LIN {X 0,Y 256.038,Z 225.896,A -85,B 0,C 180,E1 -18581.208,E2 -18581.208} C_VEL
LIN {X 0,Y 256.027,Z 225.882,A -85,B 0,C 180,E1 -18585.539,E2 -18585.539} C_VEL
LIN {X 0,Y 256.041,Z 225.899,A -85,B 0,C 180,E1 -18588.801,E2 -18588.801} C_VEL
LIN {X 0,Y 256.118,Z 225.896,A -85,B 0,C 180,E1 -18592.872,E2 -18592.872} C_VEL
LIN {X 0,Y 256.057,Z 225.889,A -85,B 0,C 180,E1 -18596.712,E2 -18596.712} C_VEL
LIN {X 0,Y 256.085,Z 225.887,A -85,B 0,C 180,E1 -18599.189,E2 -18599.189} C_VEL
LIN {X 0,Y 256.928,Z 228.457,A -85,B 0,C 180,E1 -18599.571,E2 -18599.571} C_VEL
LIN {X 0,Y 258.802,Z 230.64,A -85,B 0,C 180,E1 -18600.2,E2 -18600.2} C_VEL
LIN {X 0,Y 259.731,Z 231.462,A -85,B 0,C 180,E1 -18600.494,E2 -18600.494} C_VEL
LIN {X 0,Y 261.745,Z 234.708,A -85,B 0,C 180,E1 -18601.184,E2 -18601.184} C_VEL
LIN {X 0,Y 263.592,Z 236.729,A -85,B 0,C 180,E1 -18601.759,E2 -18601.759} C_VEL
LIN {X 0,Y 266.247,Z 240.339,A -85,B 0,C 180,E1 -18602.596,E2 -18602.596} C_VEL
LIN {X 0,Y 273.442,Z 250.412,A -85,B 0,C 180,E1 -18604.75,E2 -18604.75} C_VEL
LIN {X 0,Y 282.168,Z 263.234,A -85,B 0,C 180,E1 -18607.158,E2 -18607.158} C_VEL
LIN {X 0,Y 292.343,Z 279.507,A -85,B 0,C 180,E1 -18609.748,E2 -18609.748} C_VEL
LIN {X 0,Y 301.413,Z 295.689,A -85,B 0,C 180,E1 -18611.909,E2 -18611.909} C_VEL
LIN {X 0,Y 301.792,Z 296.477,A -85,B 0,C 180,E1 -18611.999,E2 -18611.999} C_VEL
LIN {X 0,Y 294.908,Z 420.321,A -85,B 0,C 180,E1 -18614.984,E2 -18614.984} C_VEL
LIN {X 0,Y 293.147,Z 437.641,A -85,B 0,C 180,E1 -18615.646,E2 -18615.646} C_VEL
LIN {X 0,Y 291.033,Z 452.968,A -85,B 0,C 180,E1 -18616.475,E2 -18616.475} C_VEL
LIN {X 0,Y 288.503,Z 467.873,A -85,B 0,C 180,E1 -18617.518,E2 -18617.518} C_VEL
LIN {X 0,Y 285.534,Z 482.731,A -85,B 0,C 180,E1 -18618.827,E2 -18618.827} C_VEL
LIN {X 0,Y 282.223,Z 496.554,A -85,B 0,C 180,E1 -18620.327,E2 -18620.327} C_VEL
LIN {X 0,Y 278.395,Z 510.812,A -85,B 0,C 180,E1 -18622.205,E2 -18622.205} C_VEL
LIN {X 0,Y 274.89,Z 522.936,A -85,B 0,C 180,E1 -18624.134,E2 -18624.134} C_VEL
LIN {X 0,Y 271.37,Z 534.312,A -85,B 0,C 180,E1 -18626.291,E2 -18626.291} C_VEL
LIN {X 0,Y 267.802,Z 545.342,A -85,B 0,C 180,E1 -18628.802,E2 -18628.802} C_VEL
LIN {X 0,Y 264.442,Z 555.354,A -85,B 0,C 180,E1 -18631.527,E2 -18631.527} C_VEL
LIN {X 0,Y 261.64,Z 563.721,A -85,B 0,C 180,E1 -18634.24,E2 -18634.24} C_VEL
LIN {X 0,Y 258.799,Z 572.627,A -85,B 0,C 180,E1 -18637.807,E2 -18637.807} C_VEL
LIN {X 0,Y 256.937,Z 579.031,A -85,B 0,C 180,E1 -18641.042,E2 -18641.042} C_VEL
LIN {X 0,Y 255.526,Z 584.251,A -85,B 0,C 180,E1 -18644.335,E2 -18644.335} C_VEL
LIN {X 0,Y 254.507,Z 588.356,A -85,B 0,C 180,E1 -18647.687,E2 -18647.687} C_VEL
LIN {X 0,Y 253.858,Z 591.244,A -85,B 0,C 180,E1 -18651.097,E2 -18651.097} C_VEL
LIN {X 0,Y 253.55,Z 593.058,A -85,B 0,C 180,E1 -18654.571,E2 -18654.571} C_VEL
LIN {X 0,Y 253.564,Z 593.757,A -85,B 0,C 180,E1 -18658.115,E2 -18658.115} C_VEL
LIN {X 0,Y 253.804,Z 593.171,A -85,B 0,C 180,E1 -18661.747,E2 -18661.747} C_VEL
LIN {X 0,Y 254.377,Z 591.318,A -85,B 0,C 180,E1 -18665.467,E2 -18665.467} C_VEL
LIN {X 0,Y 255.541,Z 588.082,A -85,B 0,C 180,E1 -18669.242,E2 -18669.242} C_VEL
LIN {X 0,Y 257.285,Z 583.305,A -85,B 0,C 180,E1 -18673.074,E2 -18673.074} C_VEL
LIN {X 0,Y 259.119,Z 578.582,A -85,B 0,C 180,E1 -18675.953,E2 -18675.953} C_VEL
LIN {X 0,Y 262.023,Z 571.463,A -85,B 0,C 180,E1 -18679.434,E2 -18679.434} C_VEL
LIN {X 0,Y 265.48,Z 563.42,A -85,B 0,C 180,E1 -18682.581,E2 -18682.581} C_VEL
LIN {X 0,Y 269.291,Z 554.393,A -85,B 0,C 180,E1 -18685.475,E2 -18685.475} C_VEL
LIN {X 0,Y 273.337,Z 544.565,A -85,B 0,C 180,E1 -18688.051,E2 -18688.051} C_VEL
LIN {X 0,Y 277.708,Z 533.552,A -85,B 0,C 180,E1 -18690.454,E2 -18690.454} C_VEL
LIN {X 0,Y 282.075,Z 521.913,A -85,B 0,C 180,E1 -18692.578,E2 -18692.578} C_VEL
LIN {X 0,Y 286.394,Z 509.229,A -85,B 0,C 180,E1 -18694.499,E2 -18694.499} C_VEL
LIN {X 0,Y 290.638,Z 495.548,A -85,B 0,C 180,E1 -18696.193,E2 -18696.193} C_VEL
LIN {X 0,Y 294.579,Z 480.888,A -85,B 0,C 180,E1 -18697.688,E2 -18697.688} C_VEL
LIN {X 0,Y 298.07,Z 466.156,A -85,B 0,C 180,E1 -18698.882,E2 -18698.882} C_VEL
LIN {X 0,Y 301.12,Z 449.617,A -85,B 0,C 180,E1 -18699.957,E2 -18699.957} C_VEL
LIN {X 0,Y 303.68,Z 432.171,A -85,B 0,C 180,E1 -18700.764,E2 -18700.764} C_VEL
LIN {X 0,Y 305.378,Z 415.089,A -85,B 0,C 180,E1 -18701.291,E2 -18701.291} C_VEL
LIN {X 0,Y 306.012,Z 404.805,A -85,B 0,C 180,E1 -18701.555,E2 -18701.555} C_VEL
LIN {X 0,Y 305.769,Z 400.957,A -85,B 0,C 180,E1 -18701.757,E2 -18701.757} C_VEL
LIN {X 0,Y 302.881,Z 389.177,A -85,B 0,C 180,E1 -18702.878,E2 -18702.878} C_VEL
LIN {X 0,Y 302.776,Z 385.325,A -85,B 0,C 180,E1 -18703.057,E2 -18703.057} C_VEL
LIN {X 0,Y 308.251,Z 305.412,A -85,B 0,C 180,E1 -18704.992,E2 -18704.992} C_VEL
LIN {X 0,Y 302.68,Z 295.118,A -85,B 0,C 180,E1 -18706.932,E2 -18706.932} C_VEL
LIN {X 0,Y 297.182,Z 285.913,A -85,B 0,C 180,E1 -18709.029,E2 -18709.029} C_VEL
LIN {X 0,Y 292.134,Z 278.185,A -85,B 0,C 180,E1 -18711.157,E2 -18711.157} C_VEL
LIN {X 0,Y 288.761,Z 273.365,A -85,B 0,C 180,E1 -18712.725,E2 -18712.725} C_VEL
LIN {X 0,Y 286.101,Z 269.539,A -85,B 0,C 180,E1 -18714.079,E2 -18714.079} C_VEL
LIN {X 0,Y 283.274,Z 265.593,A -85,B 0,C 180,E1 -18715.636,E2 -18715.636} C_VEL
LIN {X 0,Y 280.468,Z 261.788,A -85,B 0,C 180,E1 -18717.378,E2 -18717.378} C_VEL
LIN {X 0,Y 277.317,Z 257.984,A -85,B 0,C 180,E1 -18719.571,E2 -18719.571} C_VEL
LIN {X 0,Y 276.388,Z 256.203,A -85,B 0,C 180,E1 -18720.363,E2 -18720.363} C_VEL
LIN {X 0,Y 273.687,Z 253.629,A -85,B 0,C 180,E1 -18722.755,E2 -18722.755} C_VEL
LIN {X 0,Y 272.252,Z 251.029,A -85,B 0,C 180,E1 -18724.441,E2 -18724.441} C_VEL
LIN {X 0,Y 268.845,Z 248.558,A -85,B 0,C 180,E1 -18730.543,E2 -18730.543} C_VEL
LIN {X 0,Y 268.488,Z 248.039,A -85,B 0,C 180,E1 -18733.625,E2 -18733.625} C_VEL
LIN {X 0,Y 269.382,Z 249.399,A -85,B 0,C 180,E1 -18737.862,E2 -18737.862} C_VEL
LIN {X 0,Y 272.037,Z 251.261,A -85,B 0,C 180,E1 -18741.994,E2 -18741.994} C_VEL
LIN {X 0,Y 273.82,Z 254.481,A -85,B 0,C 180,E1 -18744.088,E2 -18744.088} C_VEL
LIN {X 0,Y 276.278,Z 256.688,A -85,B 0,C 180,E1 -18746.239,E2 -18746.239} C_VEL
LIN {X 0,Y 278.589,Z 260.18,A -85,B 0,C 180,E1 -18748.044,E2 -18748.044} C_VEL
LIN {X 0,Y 280.384,Z 262.136,A -85,B 0,C 180,E1 -18749.233,E2 -18749.233} C_VEL
LIN {X 0,Y 285.039,Z 268.873,A -85,B 0,C 180,E1 -18752.04,E2 -18752.04} C_VEL
LIN {X 0,Y 289.206,Z 275.406,A -85,B 0,C 180,E1 -18754.208,E2 -18754.208} C_VEL
LIN {X 0,Y 293.992,Z 283.483,A -85,B 0,C 180,E1 -18756.42,E2 -18756.42} C_VEL
LIN {X 0,Y 299.014,Z 292.67,A -85,B 0,C 180,E1 -18758.503,E2 -18758.503} C_VEL
LIN {X 0,Y 304.296,Z 303.274,A -85,B 0,C 180,E1 -18760.508,E2 -18760.508} C_VEL
LIN {X 0,Y 308.003,Z 311.578,A -85,B 0,C 180,E1 -18761.836,E2 -18761.836} C_VEL
LIN {X 0,Y 299.594,Z 433.298,A -85,B 0,C 180,E1 -18764.803,E2 -18764.803} C_VEL
LIN {X 0,Y 297.272,Z 451.036,A -85,B 0,C 180,E1 -18765.45,E2 -18765.45} C_VEL
LIN {X 0,Y 294.278,Z 467.286,A -85,B 0,C 180,E1 -18766.281,E2 -18766.281} C_VEL
LIN {X 0,Y 290.622,Z 483.374,A -85,B 0,C 180,E1 -18767.379,E2 -18767.379} C_VEL
LIN {X 0,Y 286.484,Z 498.911,A -85,B 0,C 180,E1 -18768.751,E2 -18768.751} C_VEL
LIN {X 0,Y 282.022,Z 513.293,A -85,B 0,C 180,E1 -18770.312,E2 -18770.312} C_VEL
LIN {X 0,Y 277.311,Z 527.146,A -85,B 0,C 180,E1 -18772.179,E2 -18772.179} C_VEL
LIN {X 0,Y 272.824,Z 538.984,A -85,B 0,C 180,E1 -18774.12,E2 -18774.12} C_VEL
LIN {X 0,Y 267.857,Z 551.328,A -85,B 0,C 180,E1 -18776.562,E2 -18776.562} C_VEL
LIN {X 0,Y 263.501,Z 561.999,A -85,B 0,C 180,E1 -18779.137,E2 -18779.137} C_VEL
LIN {X 0,Y 259.085,Z 572.215,A -85,B 0,C 180,E1 -18782.097,E2 -18782.097} C_VEL
LIN {X 0,Y 254.995,Z 581.851,A -85,B 0,C 180,E1 -18785.577,E2 -18785.577} C_VEL
LIN {X 0,Y 251.539,Z 590.511,A -85,B 0,C 180,E1 -18789.555,E2 -18789.555} C_VEL
LIN {X 0,Y 249.159,Z 597.289,A -85,B 0,C 180,E1 -18793.613,E2 -18793.613} C_VEL
LIN {X 0,Y 247.861,Z 601.425,A -85,B 0,C 180,E1 -18796.886,E2 -18796.886} C_VEL
LIN {X 0,Y 247.112,Z 604.608,A -85,B 0,C 180,E1 -18800.171,E2 -18800.171} C_VEL
LIN {X 0,Y 246.859,Z 606.706,A -85,B 0,C 180,E1 -18803.457,E2 -18803.457} C_VEL
LIN {X 0,Y 246.839,Z 607.901,A -85,B 0,C 180,E1 -18806.732,E2 -18806.732} C_VEL
LIN {X 0,Y 246.982,Z 608.041,A -85,B 0,C 180,E1 -18809.996,E2 -18809.996} C_VEL
LIN {X 0,Y 246.867,Z 607.256,A -85,B 0,C 180,E1 -18813.26,E2 -18813.26} C_VEL
LIN {X 0,Y 246.908,Z 606.416,A -85,B 0,C 180,E1 -18814.977,E2 -18814.977} C_VEL
LIN {X 0,Y 246.951,Z 604.091,A -85,B 0,C 180,E1 -18818.176,E2 -18818.176} C_VEL
LIN {X 0,Y 247.356,Z 600.725,A -85,B 0,C 180,E1 -18821.467,E2 -18821.467} C_VEL
LIN {X 0,Y 248.35,Z 596.177,A -85,B 0,C 180,E1 -18824.751,E2 -18824.751} C_VEL
LIN {X 0,Y 249.763,Z 590.504,A -85,B 0,C 180,E1 -18828.026,E2 -18828.026} C_VEL
LIN {X 0,Y 251.845,Z 583.51,A -85,B 0,C 180,E1 -18831.266,E2 -18831.266} C_VEL
LIN {X 0,Y 254.487,Z 575.039,A -85,B 0,C 180,E1 -18834.467,E2 -18834.467} C_VEL
LIN {X 0,Y 257.909,Z 564.935,A -85,B 0,C 180,E1 -18837.592,E2 -18837.592} C_VEL
LIN {X 0,Y 261.447,Z 554.509,A -85,B 0,C 180,E1 -18840.261,E2 -18840.261} C_VEL
LIN {X 0,Y 264.867,Z 544.091,A -85,B 0,C 180,E1 -18842.495,E2 -18842.495} C_VEL
LIN {X 0,Y 268.706,Z 531.999,A -85,B 0,C 180,E1 -18844.666,E2 -18844.666} C_VEL
LIN {X 0,Y 272.764,Z 518.677,A -85,B 0,C 180,E1 -18846.641,E2 -18846.641} C_VEL
LIN {X 0,Y 276.338,Z 505.257,A -85,B 0,C 180,E1 -18848.304,E2 -18848.304} C_VEL
LIN {X 0,Y 280.028,Z 490.239,A -85,B 0,C 180,E1 -18849.784,E2 -18849.784} C_VEL
LIN {X 0,Y 283.164,Z 474.912,A -85,B 0,C 180,E1 -18851.002,E2 -18851.002} C_VEL
LIN {X 0,Y 285.87,Z 458.777,A -85,B 0,C 180,E1 -18851.996,E2 -18851.996} C_VEL
LIN {X 0,Y 288.082,Z 442.453,A -85,B 0,C 180,E1 -18852.721,E2 -18852.721} C_VEL
LIN {X 0,Y 289.436,Z 426.385,A -85,B 0,C 180,E1 -18853.222,E2 -18853.222} C_VEL
LIN {X 0,Y 296.146,Z 306.323,A -85,B 0,C 180,E1 -18856.146,E2 -18856.146} C_VEL
LIN {X 0,Y 288.318,Z 289.97,A -85,B 0,C 180,E1 -18858.143,E2 -18858.143} C_VEL
LIN {X 0,Y 280.841,Z 275.817,A -85,B 0,C 180,E1 -18860.152,E2 -18860.152} C_VEL
LIN {X 0,Y 272.784,Z 261.806,A -85,B 0,C 180,E1 -18862.449,E2 -18862.449} C_VEL
LIN {X 0,Y 263.31,Z 246.71,A -85,B 0,C 180,E1 -18865.389,E2 -18865.389} C_VEL
LIN {X 0,Y 259.388,Z 241.321,A -85,B 0,C 180,E1 -18866.667,E2 -18866.667} C_VEL
LIN {X 0,Y 256.72,Z 237.707,A -85,B 0,C 180,E1 -18867.574,E2 -18867.574} C_VEL
LIN {X 0,Y 253.409,Z 233.62,A -85,B 0,C 180,E1 -18868.726,E2 -18868.726} C_VEL
LIN {X 0,Y 252.392,Z 231.94,A -85,B 0,C 180,E1 -18869.11,E2 -18869.11} C_VEL
LIN {X 0,Y 250.174,Z 229.865,A -85,B 0,C 180,E1 -18869.889,E2 -18869.889} C_VEL
LIN {X 0,Y 249.156,Z 227.398,A -85,B 0,C 180,E1 -18870.335,E2 -18870.335} C_VEL
LIN {X 0,Y 249.056,Z 226.774,A -85,B 0,C 180,E1 -18870.427,E2 -18870.427} C_VEL
LIN {X 0,Y 249.129,Z 226.741,A -85,B 0,C 180,E1 -18874.967,E2 -18874.967} C_VEL
LIN {X 0,Y 249.109,Z 226.742,A -85,B 0,C 180,E1 -18878.577,E2 -18878.577} C_VEL
LIN {X 0,Y 249.217,Z 226.755,A -85,B 0,C 180,E1 -18883.621,E2 -18883.621} C_VEL
LIN {X 0,Y 249.226,Z 226.706,A -85,B 0,C 180,E1 -18888.616,E2 -18888.616} C_VEL
LIN {X 0,Y 249.453,Z 226.725,A -85,B 0,C 180,E1 -18891.903,E2 -18891.903} C_VEL
LIN {X 0,Y 249.406,Z 226.675,A -85,B 0,C 180,E1 -18896.77,E2 -18896.77} C_VEL
LIN {X 0,Y 249.701,Z 226.689,A -85,B 0,C 180,E1 -18900.001,E2 -18900.001} C_VEL
LIN {X 0,Y 249.406,Z 226.706,A -85,B 0,C 180,E1 -18903.232,E2 -18903.232} C_VEL
LIN {X 0,Y 249.411,Z 226.715,A -85,B 0,C 180,E1 -18906.78,E2 -18906.78} C_VEL
LIN {X 0,Y 249.318,Z 226.724,A -85,B 0,C 180,E1 -18909.738,E2 -18909.738} C_VEL
LIN {X 0,Y 249.176,Z 226.755,A -85,B 0,C 180,E1 -18914.706,E2 -18914.706} C_VEL
LIN {X 0,Y 249.115,Z 226.735,A -85,B 0,C 180,E1 -18918.08,E2 -18918.08} C_VEL
LIN {X 0,Y 249.065,Z 226.767,A -85,B 0,C 180,E1 -18921.521,E2 -18921.521} C_VEL
LIN {X 0,Y 249.109,Z 226.736,A -85,B 0,C 180,E1 -18925.485,E2 -18925.485} C_VEL
LIN {X 0,Y 249.063,Z 226.773,A -85,B 0,C 180,E1 -18928.997,E2 -18928.997} C_VEL
LIN {X 0,Y 249.011,Z 226.751,A -85,B 0,C 180,E1 -18932.43,E2 -18932.43} C_VEL
LIN {X 0,Y 249.029,Z 226.778,A -85,B 0,C 180,E1 -18936.347,E2 -18936.347} C_VEL
LIN {X 0,Y 248.976,Z 226.764,A -85,B 0,C 180,E1 -18940.485,E2 -18940.485} C_VEL
LIN {X 0,Y 248.986,Z 226.782,A -85,B 0,C 180,E1 -18942.795,E2 -18942.795} C_VEL
LIN {X 0,Y 248.996,Z 226.78,A -85,B 0,C 180,E1 -18947.366,E2 -18947.366} C_VEL
LIN {X 0,Y 249.032,Z 226.769,A -85,B 0,C 180,E1 -18952.205,E2 -18952.205} C_VEL
LIN {X 0,Y 249.031,Z 226.763,A -85,B 0,C 180,E1 -18956.618,E2 -18956.618} C_VEL
LIN {X 0,Y 249.009,Z 226.772,A -85,B 0,C 180,E1 -18957.093,E2 -18957.093} C_VEL
LIN {X 0,Y 249.907,Z 229.476,A -85,B 0,C 180,E1 -18957.532,E2 -18957.532} C_VEL
LIN {X 0,Y 251.995,Z 231.702,A -85,B 0,C 180,E1 -18958.28,E2 -18958.28} C_VEL
LIN {X 0,Y 252.914,Z 232.566,A -85,B 0,C 180,E1 -18958.598,E2 -18958.598} C_VEL
LIN {X 0,Y 254.905,Z 235.733,A -85,B 0,C 180,E1 -18959.339,E2 -18959.339} C_VEL
LIN {X 0,Y 256.628,Z 237.548,A -85,B 0,C 180,E1 -18959.919,E2 -18959.919} C_VEL
LIN {X 0,Y 259.169,Z 241.121,A -85,B 0,C 180,E1 -18960.789,E2 -18960.789} C_VEL
LIN {X 0,Y 260.595,Z 242.915,A -85,B 0,C 180,E1 -18961.253,E2 -18961.253} C_VEL
LIN {X 0,Y 267.808,Z 252.881,A -85,B 0,C 180,E1 -18963.525,E2 -18963.525} C_VEL
LIN {X 0,Y 277.279,Z 266.774,A -85,B 0,C 180,E1 -18966.261,E2 -18966.261} C_VEL
LIN {X 0,Y 287.941,Z 283.964,A -85,B 0,C 180,E1 -18969.081,E2 -18969.081} C_VEL
LIN {X 0,Y 296.28,Z 298.863,A -85,B 0,C 180,E1 -18971.129,E2 -18971.129} C_VEL
LIN {X 0,Y 289.398,Z 420.084,A -85,B 0,C 180,E1 -18974.104,E2 -18974.104} C_VEL
LIN {X 0,Y 287.7,Z 436.638,A -85,B 0,C 180,E1 -18974.734,E2 -18974.734} C_VEL
LIN {X 0,Y 285.512,Z 452.308,A -85,B 0,C 180,E1 -18975.572,E2 -18975.572} C_VEL
LIN {X 0,Y 282.695,Z 468.412,A -85,B 0,C 180,E1 -18976.709,E2 -18976.709} C_VEL
LIN {X 0,Y 279.498,Z 483.759,A -85,B 0,C 180,E1 -18978.093,E2 -18978.093} C_VEL
LIN {X 0,Y 276.228,Z 496.992,A -85,B 0,C 180,E1 -18979.56,E2 -18979.56} C_VEL
LIN {X 0,Y 272.277,Z 511.211,A -85,B 0,C 180,E1 -18981.469,E2 -18981.469} C_VEL
LIN {X 0,Y 268.088,Z 524.98,A -85,B 0,C 180,E1 -18983.734,E2 -18983.734} C_VEL
LIN {X 0,Y 264.114,Z 537.241,A -85,B 0,C 180,E1 -18986.189,E2 -18986.189} C_VEL
LIN {X 0,Y 260.375,Z 548.339,A -85,B 0,C 180,E1 -18988.873,E2 -18988.873} C_VEL
LIN {X 0,Y 256.717,Z 558.837,A -85,B 0,C 180,E1 -18991.965,E2 -18991.965} C_VEL
LIN {X 0,Y 253.366,Z 568.512,A -85,B 0,C 180,E1 -18995.495,E2 -18995.495} C_VEL
LIN {X 0,Y 250.967,Z 575.869,A -85,B 0,C 180,E1 -18998.864,E2 -18998.864} C_VEL
LIN {X 0,Y 249.226,Z 581.744,A -85,B 0,C 180,E1 -19002.213,E2 -19002.213} C_VEL
LIN {X 0,Y 248.035,Z 586.383,A -85,B 0,C 180,E1 -19005.55,E2 -19005.55} C_VEL
LIN {X 0,Y 247.278,Z 589.203,A -85,B 0,C 180,E1 -19008.222,E2 -19008.222} C_VEL
LIN {X 0,Y 246.668,Z 591.951,A -85,B 0,C 180,E1 -19011.743,E2 -19011.743} C_VEL
LIN {X 0,Y 246.429,Z 593.489,A -85,B 0,C 180,E1 -19015.331,E2 -19015.331} C_VEL
LIN {X 0,Y 246.496,Z 593.914,A -85,B 0,C 180,E1 -19018.996,E2 -19018.996} C_VEL
LIN {X 0,Y 246.813,Z 593.149,A -85,B 0,C 180,E1 -19022.757,E2 -19022.757} C_VEL
LIN {X 0,Y 247.57,Z 591.009,A -85,B 0,C 180,E1 -19026.598,E2 -19026.598} C_VEL
LIN {X 0,Y 248.959,Z 587.441,A -85,B 0,C 180,E1 -19030.49,E2 -19030.49} C_VEL
LIN {X 0,Y 250.174,Z 584.29,A -85,B 0,C 180,E1 -19033.078,E2 -19033.078} C_VEL
LIN {X 0,Y 252.3,Z 579.106,A -85,B 0,C 180,E1 -19036.41,E2 -19036.41} C_VEL
LIN {X 0,Y 255.24,Z 572.41,A -85,B 0,C 180,E1 -19039.829,E2 -19039.829} C_VEL
LIN {X 0,Y 258.535,Z 565.201,A -85,B 0,C 180,E1 -19042.801,E2 -19042.801} C_VEL
LIN {X 0,Y 262.429,Z 556.354,A -85,B 0,C 180,E1 -19045.778,E2 -19045.778} C_VEL
LIN {X 0,Y 266.526,Z 547.015,A -85,B 0,C 180,E1 -19048.381,E2 -19048.381} C_VEL
LIN {X 0,Y 270.957,Z 536.584,A -85,B 0,C 180,E1 -19050.81,E2 -19050.81} C_VEL
LIN {X 0,Y 275.696,Z 524.377,A -85,B 0,C 180,E1 -19053.156,E2 -19053.156} C_VEL
LIN {X 0,Y 280.55,Z 511.023,A -85,B 0,C 180,E1 -19055.246,E2 -19055.246} C_VEL
LIN {X 0,Y 284.791,Z 498.12,A -85,B 0,C 180,E1 -19056.909,E2 -19056.909} C_VEL
LIN {X 0,Y 288.97,Z 483.644,A -85,B 0,C 180,E1 -19058.454,E2 -19058.454} C_VEL
LIN {X 0,Y 292.841,Z 468.101,A -85,B 0,C 180,E1 -19059.769,E2 -19059.769} C_VEL
LIN {X 0,Y 295.961,Z 452.361,A -85,B 0,C 180,E1 -19060.821,E2 -19060.821} C_VEL
LIN {X 0,Y 298.537,Z 435.936,A -85,B 0,C 180,E1 -19061.641,E2 -19061.641} C_VEL
LIN {X 0,Y 300.516,Z 418.44,A -85,B 0,C 180,E1 -19062.234,E2 -19062.234} C_VEL
LIN {X 0,Y 302.776,Z 385.325,A -85,B 0,C 180,E1 -19063.057,E2 -19063.057} C_VEL
LIN {X 0,Y 302.834,Z 379.541,A -85,B 0,C 180,E1 -19063.278,E2 -19063.278} C_VEL
LIN {X 0,Y 301.699,Z 370.313,A -85,B 0,C 180,E1 -19063.936,E2 -19063.936} C_VEL
LIN {X 0,Y 300.552,Z 361.092,A -85,B 0,C 180,E1 -19064.612,E2 -19064.612} C_VEL
LIN {X 0,Y 300.563,Z 355.31,A -85,B 0,C 180,E1 -19064.855,E2 -19064.855} C_VEL
LIN {X 0,Y 303.884,Z 308.521,A -85,B 0,C 180,E1 -19066.007,E2 -19066.007} C_VEL
LIN {X 0,Y 298.074,Z 297.794,A -85,B 0,C 180,E1 -19068.171,E2 -19068.171} C_VEL
LIN {X 0,Y 293.131,Z 289.563,A -85,B 0,C 180,E1 -19070.187,E2 -19070.187} C_VEL
LIN {X 0,Y 289.122,Z 283.386,A -85,B 0,C 180,E1 -19071.983,E2 -19071.983} C_VEL
LIN {X 0,Y 284.509,Z 276.454,A -85,B 0,C 180,E1 -19074.329,E2 -19074.329} C_VEL
LIN {X 0,Y 281.361,Z 272.03,A -85,B 0,C 180,E1 -19076.125,E2 -19076.125} C_VEL
LIN {X 0,Y 278.07,Z 267.628,A -85,B 0,C 180,E1 -19078.261,E2 -19078.261} C_VEL
LIN {X 0,Y 275.471,Z 264.089,A -85,B 0,C 180,E1 -19080.228,E2 -19080.228} C_VEL
LIN {X 0,Y 274.706,Z 262.786,A -85,B 0,C 180,E1 -19080.915,E2 -19080.915} C_VEL
LIN {X 0,Y 272.3,Z 260.326,A -85,B 0,C 180,E1 -19083.154,E2 -19083.154} C_VEL
LIN {X 0,Y 271.101,Z 258.011,A -85,B 0,C 180,E1 -19084.646,E2 -19084.646} C_VEL
LIN {X 0,Y 267.875,Z 255.592,A -85,B 0,C 180,E1 -19090.582,E2 -19090.582} C_VEL
LIN {X 0,Y 267.54,Z 255.058,A -85,B 0,C 180,E1 -19093.675,E2 -19093.675} C_VEL
LIN {X 0,Y 269.01,Z 256.997,A -85,B 0,C 180,E1 -19099.06,E2 -19099.06} C_VEL
LIN {X 0,Y 270.831,Z 258.241,A -85,B 0,C 180,E1 -19101.721,E2 -19101.721} C_VEL
LIN {X 0,Y 272.644,Z 261.462,A -85,B 0,C 180,E1 -19103.918,E2 -19103.918} C_VEL
LIN {X 0,Y 274.806,Z 263.495,A -85,B 0,C 180,E1 -19105.865,E2 -19105.865} C_VEL
LIN {X 0,Y 277.37,Z 267.233,A -85,B 0,C 180,E1 -19107.919,E2 -19107.919} C_VEL
LIN {X 0,Y 278.726,Z 268.794,A -85,B 0,C 180,E1 -19108.842,E2 -19108.842} C_VEL
LIN {X 0,Y 283.026,Z 275.276,A -85,B 0,C 180,E1 -19111.553,E2 -19111.553} C_VEL
LIN {X 0,Y 287.145,Z 281.958,A -85,B 0,C 180,E1 -19113.772,E2 -19113.772} C_VEL
LIN {X 0,Y 291.968,Z 290.428,A -85,B 0,C 180,E1 -19116.085,E2 -19116.085} C_VEL
LIN {X 0,Y 297.475,Z 300.983,A -85,B 0,C 180,E1 -19118.432,E2 -19118.432} C_VEL
LIN {X 0,Y 302.651,Z 312.143,A -85,B 0,C 180,E1 -19120.45,E2 -19120.45} C_VEL
LIN {X 0,Y 303.684,Z 314.617,A -85,B 0,C 180,E1 -19120.838,E2 -19120.838} C_VEL
LIN {X 0,Y 295.081,Z 433.216,A -85,B 0,C 180,E1 -19123.744,E2 -19123.744} C_VEL
LIN {X 0,Y 292.778,Z 450.274,A -85,B 0,C 180,E1 -19124.364,E2 -19124.364} C_VEL
LIN {X 0,Y 289.776,Z 466.339,A -85,B 0,C 180,E1 -19125.179,E2 -19125.179} C_VEL
LIN {X 0,Y 285.978,Z 482.599,A -85,B 0,C 180,E1 -19126.274,E2 -19126.274} C_VEL
LIN {X 0,Y 282.19,Z 496.689,A -85,B 0,C 180,E1 -19127.5,E2 -19127.5} C_VEL
LIN {X 0,Y 277.537,Z 511.374,A -85,B 0,C 180,E1 -19129.061,E2 -19129.061} C_VEL
LIN {X 0,Y 272.87,Z 524.548,A -85,B 0,C 180,E1 -19130.81,E2 -19130.81} C_VEL
LIN {X 0,Y 267.863,Z 537.438,A -85,B 0,C 180,E1 -19132.879,E2 -19132.879} C_VEL
LIN {X 0,Y 263.374,Z 548.377,A -85,B 0,C 180,E1 -19134.987,E2 -19134.987} C_VEL
LIN {X 0,Y 258.621,Z 559.277,A -85,B 0,C 180,E1 -19137.535,E2 -19137.535} C_VEL
LIN {X 0,Y 254.368,Z 568.668,A -85,B 0,C 180,E1 -19140.174,E2 -19140.174} C_VEL
LIN {X 0,Y 250.23,Z 577.854,A -85,B 0,C 180,E1 -19143.293,E2 -19143.293} C_VEL
LIN {X 0,Y 246.892,Z 585.568,A -85,B 0,C 180,E1 -19146.511,E2 -19146.511} C_VEL
LIN {X 0,Y 244.201,Z 591.949,A -85,B 0,C 180,E1 -19149.793,E2 -19149.793} C_VEL
LIN {X 0,Y 242.221,Z 597.355,A -85,B 0,C 180,E1 -19153.231,E2 -19153.231} C_VEL
LIN {X 0,Y 240.88,Z 601.326,A -85,B 0,C 180,E1 -19156.498,E2 -19156.498} C_VEL
LIN {X 0,Y 240.049,Z 604.468,A -85,B 0,C 180,E1 -19159.879,E2 -19159.879} C_VEL
LIN {X 0,Y 239.77,Z 606.548,A -85,B 0,C 180,E1 -19163.263,E2 -19163.263} C_VEL
LIN {X 0,Y 239.744,Z 607.704,A -85,B 0,C 180,E1 -19166.635,E2 -19166.635} C_VEL
LIN {X 0,Y 239.912,Z 607.825,A -85,B 0,C 180,E1 -19169.996,E2 -19169.996} C_VEL
LIN {X 0,Y 239.773,Z 606.999,A -85,B 0,C 180,E1 -19173.357,E2 -19173.357} C_VEL
LIN {X 0,Y 239.817,Z 606.2,A -85,B 0,C 180,E1 -19175.04,E2 -19175.04} C_VEL
LIN {X 0,Y 239.869,Z 603.79,A -85,B 0,C 180,E1 -19178.42,E2 -19178.42} C_VEL
LIN {X 0,Y 240.328,Z 600.398,A -85,B 0,C 180,E1 -19181.808,E2 -19181.808} C_VEL
LIN {X 0,Y 241.667,Z 594.763,A -85,B 0,C 180,E1 -19185.876,E2 -19185.876} C_VEL
LIN {X 0,Y 243.368,Z 588.425,A -85,B 0,C 180,E1 -19189.391,E2 -19189.391} C_VEL
LIN {X 0,Y 245.761,Z 581.043,A -85,B 0,C 180,E1 -19192.704,E2 -19192.704} C_VEL
LIN {X 0,Y 248.755,Z 572.18,A -85,B 0,C 180,E1 -19195.966,E2 -19195.966} C_VEL
LIN {X 0,Y 252.554,Z 561.576,A -85,B 0,C 180,E1 -19199.137,E2 -19199.137} C_VEL
LIN {X 0,Y 256.203,Z 550.95,A -85,B 0,C 180,E1 -19201.749,E2 -19201.749} C_VEL
LIN {X 0,Y 260.116,Z 539.507,A -85,B 0,C 180,E1 -19204.094,E2 -19204.094} C_VEL
LIN {X 0,Y 264.255,Z 526.727,A -85,B 0,C 180,E1 -19206.275,E2 -19206.275} C_VEL
LIN {X 0,Y 268.286,Z 513.067,A -85,B 0,C 180,E1 -19208.199,E2 -19208.199} C_VEL
LIN {X 0,Y 272.426,Z 497.808,A -85,B 0,C 180,E1 -19209.914,E2 -19209.914} C_VEL
LIN {X 0,Y 275.764,Z 483.143,A -85,B 0,C 180,E1 -19211.25,E2 -19211.25} C_VEL
LIN {X 0,Y 278.855,Z 467.321,A -85,B 0,C 180,E1 -19212.384,E2 -19212.384} C_VEL
LIN {X 0,Y 281.427,Z 451.327,A -85,B 0,C 180,E1 -19213.244,E2 -19213.244} C_VEL
LIN {X 0,Y 283.433,Z 434.03,A -85,B 0,C 180,E1 -19213.902,E2 -19213.902} C_VEL
LIN {X 0,Y 290.792,Z 308.784,A -85,B 0,C 180,E1 -19217.015,E2 -19217.015} C_VEL
LIN {X 0,Y 283.393,Z 293.31,A -85,B 0,C 180,E1 -19218.974,E2 -19218.974} C_VEL
LIN {X 0,Y 276.255,Z 279.762,A -85,B 0,C 180,E1 -19220.962,E2 -19220.962} C_VEL
LIN {X 0,Y 269.016,Z 266.93,A -85,B 0,C 180,E1 -19223.113,E2 -19223.113} C_VEL
LIN {X 0,Y 259.944,Z 252.291,A -85,B 0,C 180,E1 -19226.014,E2 -19226.014} C_VEL
LIN {X 0,Y 256.068,Z 246.936,A -85,B 0,C 180,E1 -19227.318,E2 -19227.318} C_VEL
LIN {X 0,Y 252.602,Z 242.357,A -85,B 0,C 180,E1 -19228.532,E2 -19228.532} C_VEL
LIN {X 0,Y 249.969,Z 238.83,A -85,B 0,C 180,E1 -19229.494,E2 -19229.494} C_VEL
LIN {X 0,Y 249.067,Z 237.747,A -85,B 0,C 180,E1 -19229.827,E2 -19229.827} C_VEL
LIN {X 0,Y 246.745,Z 234.989,A -85,B 0,C 180,E1 -19230.707,E2 -19230.707} C_VEL
LIN {X 0,Y 245.548,Z 232.939,A -85,B 0,C 180,E1 -19231.203,E2 -19231.203} C_VEL
LIN {X 0,Y 243.167,Z 230.76,A -85,B 0,C 180,E1 -19232.106,E2 -19232.106} C_VEL
LIN {X 0,Y 242.09,Z 228.145,A -85,B 0,C 180,E1 -19232.617,E2 -19232.617} C_VEL
LIN {X 0,Y 242.009,Z 227.625,A -85,B 0,C 180,E1 -19232.724,E2 -19232.724} C_VEL
LIN {X 0,Y 242.045,Z 227.639,A -85,B 0,C 180,E1 -19236.016,E2 -19236.016} C_VEL
LIN {X 0,Y 242.047,Z 227.609,A -85,B 0,C 180,E1 -19239.61,E2 -19239.61} C_VEL
LIN {X 0,Y 242.138,Z 227.633,A -85,B 0,C 180,E1 -19243.277,E2 -19243.277} C_VEL
LIN {X 0,Y 242.159,Z 227.584,A -85,B 0,C 180,E1 -19248.279,E2 -19248.279} C_VEL
LIN {X 0,Y 242.4,Z 227.604,A -85,B 0,C 180,E1 -19251.665,E2 -19251.665} C_VEL
LIN {X 0,Y 242.229,Z 227.575,A -85,B 0,C 180,E1 -19255.007,E2 -19255.007} C_VEL
LIN {X 0,Y 242.609,Z 227.538,A -85,B 0,C 180,E1 -19258.341,E2 -19258.341} C_VEL
LIN {X 0,Y 242.609,Z 227.576,A -85,B 0,C 180,E1 -19261.661,E2 -19261.661} C_VEL
LIN {X 0,Y 242.39,Z 227.591,A -85,B 0,C 180,E1 -19266.755,E2 -19266.755} C_VEL
LIN {X 0,Y 242.241,Z 227.6,A -85,B 0,C 180,E1 -19270.026,E2 -19270.026} C_VEL
LIN {X 0,Y 242.139,Z 227.634,A -85,B 0,C 180,E1 -19275.143,E2 -19275.143} C_VEL
LIN {X 0,Y 242.049,Z 227.612,A -85,B 0,C 180,E1 -19278.627,E2 -19278.627} C_VEL
LIN {X 0,Y 241.991,Z 227.652,A -85,B 0,C 180,E1 -19282.183,E2 -19282.183} C_VEL
LIN {X 0,Y 242.046,Z 227.614,A -85,B 0,C 180,E1 -19285.841,E2 -19285.841} C_VEL
LIN {X 0,Y 242.01,Z 227.652,A -85,B 0,C 180,E1 -19289.584,E2 -19289.584} C_VEL
LIN {X 0,Y 241.962,Z 227.629,A -85,B 0,C 180,E1 -19293.497,E2 -19293.497} C_VEL
LIN {X 0,Y 241.971,Z 227.641,A -85,B 0,C 180,E1 -19297.586,E2 -19297.586} C_VEL
LIN {X 0,Y 241.914,Z 227.663,A -85,B 0,C 180,E1 -19301.929,E2 -19301.929} C_VEL
LIN {X 0,Y 241.912,Z 227.648,A -85,B 0,C 180,E1 -19306.578,E2 -19306.578} C_VEL
LIN {X 0,Y 241.984,Z 227.639,A -85,B 0,C 180,E1 -19311.645,E2 -19311.645} C_VEL
LIN {X 0,Y 242.021,Z 227.705,A -85,B 0,C 180,E1 -19314.847,E2 -19314.847} C_VEL
LIN {X 0,Y 242.754,Z 230.068,A -85,B 0,C 180,E1 -19315.234,E2 -19315.234} C_VEL
LIN {X 0,Y 244.716,Z 232.402,A -85,B 0,C 180,E1 -19316.026,E2 -19316.026} C_VEL
LIN {X 0,Y 245.884,Z 233.353,A -85,B 0,C 180,E1 -19316.461,E2 -19316.461} C_VEL
LIN {X 0,Y 247.86,Z 236.577,A -85,B 0,C 180,E1 -19317.261,E2 -19317.261} C_VEL
LIN {X 0,Y 249.976,Z 238.735,A -85,B 0,C 180,E1 -19318.024,E2 -19318.024} C_VEL
LIN {X 0,Y 252.42,Z 242.176,A -85,B 0,C 180,E1 -19318.928,E2 -19318.928} C_VEL
LIN {X 0,Y 253.637,Z 243.686,A -85,B 0,C 180,E1 -19319.358,E2 -19319.358} C_VEL
LIN {X 0,Y 257.945,Z 249.524,A -85,B 0,C 180,E1 -19320.846,E2 -19320.846} C_VEL
LIN {X 0,Y 265.737,Z 260.308,A -85,B 0,C 180,E1 -19323.336,E2 -19323.336} C_VEL
LIN {X 0,Y 275.701,Z 275.457,A -85,B 0,C 180,E1 -19326.263,E2 -19326.263} C_VEL
LIN {X 0,Y 284.593,Z 290.161,A -85,B 0,C 180,E1 -19328.658,E2 -19328.658} C_VEL
LIN {X 0,Y 290.883,Z 301.52,A -85,B 0,C 180,E1 -19330.258,E2 -19330.258} C_VEL
LIN {X 0,Y 283.854,Z 421.067,A -85,B 0,C 180,E1 -19333.23,E2 -19333.23} C_VEL
LIN {X 0,Y 281.972,Z 438.281,A -85,B 0,C 180,E1 -19333.906,E2 -19333.906} C_VEL
LIN {X 0,Y 279.64,Z 454.169,A -85,B 0,C 180,E1 -19334.797,E2 -19334.797} C_VEL
LIN {X 0,Y 276.935,Z 468.92,A -85,B 0,C 180,E1 -19335.866,E2 -19335.866} C_VEL
LIN {X 0,Y 273.685,Z 484.087,A -85,B 0,C 180,E1 -19337.257,E2 -19337.257} C_VEL
LIN {X 0,Y 269.875,Z 498.895,A -85,B 0,C 180,E1 -19338.931,E2 -19338.931} C_VEL
LIN {X 0,Y 265.826,Z 512.816,A -85,B 0,C 180,E1 -19340.877,E2 -19340.877} C_VEL
LIN {X 0,Y 262.052,Z 524.774,A -85,B 0,C 180,E1 -19342.896,E2 -19342.896} C_VEL
LIN {X 0,Y 258.049,Z 536.754,A -85,B 0,C 180,E1 -19345.317,E2 -19345.317} C_VEL
LIN {X 0,Y 254.158,Z 547.847,A -85,B 0,C 180,E1 -19348.023,E2 -19348.023} C_VEL
LIN {X 0,Y 250.72,Z 557.26,A -85,B 0,C 180,E1 -19350.807,E2 -19350.807} C_VEL
LIN {X 0,Y 247.453,Z 566.186,A -85,B 0,C 180,E1 -19353.983,E2 -19353.983} C_VEL
LIN {X 0,Y 244.75,Z 574.057,A -85,B 0,C 180,E1 -19357.428,E2 -19357.428} C_VEL
LIN {X 0,Y 242.718,Z 580.548,A -85,B 0,C 180,E1 -19360.97,E2 -19360.97} C_VEL
LIN {X 0,Y 241.042,Z 586.468,A -85,B 0,C 180,E1 -19365.217,E2 -19365.217} C_VEL
LIN {X 0,Y 240.074,Z 590.035,A -85,B 0,C 180,E1 -19368.788,E2 -19368.788} C_VEL
LIN {X 0,Y 239.484,Z 592.525,A -85,B 0,C 180,E1 -19372.43,E2 -19372.43} C_VEL
LIN {X 0,Y 239.321,Z 593.918,A -85,B 0,C 180,E1 -19376.139,E2 -19376.139} C_VEL
LIN {X 0,Y 239.408,Z 594.163,A -85,B 0,C 180,E1 -19378.274,E2 -19378.274} C_VEL
LIN {X 0,Y 239.638,Z 593.689,A -85,B 0,C 180,E1 -19381.867,E2 -19381.867} C_VEL
LIN {X 0,Y 240.279,Z 591.979,A -85,B 0,C 180,E1 -19385.805,E2 -19385.805} C_VEL
LIN {X 0,Y 241.549,Z 588.893,A -85,B 0,C 180,E1 -19389.803,E2 -19389.803} C_VEL
LIN {X 0,Y 243.465,Z 584.324,A -85,B 0,C 180,E1 -19393.807,E2 -19393.807} C_VEL
LIN {X 0,Y 245.711,Z 579.198,A -85,B 0,C 180,E1 -19397.155,E2 -19397.155} C_VEL
LIN {X 0,Y 249.06,Z 572.003,A -85,B 0,C 180,E1 -19400.867,E2 -19400.867} C_VEL
LIN {X 0,Y 253.171,Z 563.455,A -85,B 0,C 180,E1 -19404.34,E2 -19404.34} C_VEL
LIN {X 0,Y 257.12,Z 555.066,A -85,B 0,C 180,E1 -19407.134,E2 -19407.134} C_VEL
LIN {X 0,Y 261.858,Z 544.689,A -85,B 0,C 180,E1 -19409.95,E2 -19409.95} C_VEL
LIN {X 0,Y 266.613,Z 533.65,A -85,B 0,C 180,E1 -19412.422,E2 -19412.422} C_VEL
LIN {X 0,Y 271.459,Z 521.662,A -85,B 0,C 180,E1 -19414.643,E2 -19414.643} C_VEL
LIN {X 0,Y 276.464,Z 508.23,A -85,B 0,C 180,E1 -19416.687,E2 -19416.687} C_VEL
LIN {X 0,Y 280.777,Z 495.072,A -85,B 0,C 180,E1 -19418.323,E2 -19418.323} C_VEL
LIN {X 0,Y 284.929,Z 480.634,A -85,B 0,C 180,E1 -19419.798,E2 -19419.798} C_VEL
LIN {X 0,Y 288.782,Z 465.137,A -85,B 0,C 180,E1 -19421.051,E2 -19421.051} C_VEL
LIN {X 0,Y 291.922,Z 449.395,A -85,B 0,C 180,E1 -19422.056,E2 -19422.056} C_VEL
LIN {X 0,Y 294.606,Z 432.057,A -85,B 0,C 180,E1 -19422.857,E2 -19422.857} C_VEL
LIN {X 0,Y 296.341,Z 415.218,A -85,B 0,C 180,E1 -19423.384,E2 -19423.384} C_VEL
LIN {X 0,Y 300.563,Z 355.31,A -85,B 0,C 180,E1 -19424.855,E2 -19424.855} C_VEL
LIN {X 0,Y 300.598,Z 349.537,A -85,B 0,C 180,E1 -19425.095,E2 -19425.095} C_VEL
LIN {X 0,Y 298.625,Z 331.098,A -85,B 0,C 180,E1 -19426.445,E2 -19426.445} C_VEL
LIN {X 0,Y 298.706,Z 325.325,A -85,B 0,C 180,E1 -19426.684,E2 -19426.684} C_VEL
LIN {X 0,Y 299.684,Z 311.9,A -85,B 0,C 180,E1 -19427.022,E2 -19427.022} C_VEL
LIN {X 0,Y 293.527,Z 300.43,A -85,B 0,C 180,E1 -19429.483,E2 -19429.483} C_VEL
LIN {X 0,Y 287.809,Z 290.961,A -85,B 0,C 180,E1 -19432.049,E2 -19432.049} C_VEL
LIN {X 0,Y 282.215,Z 282.466,A -85,B 0,C 180,E1 -19434.964,E2 -19434.964} C_VEL
LIN {X 0,Y 279.43,Z 278.407,A -85,B 0,C 180,E1 -19436.645,E2 -19436.645} C_VEL
LIN {X 0,Y 276.483,Z 274.31,A -85,B 0,C 180,E1 -19438.634,E2 -19438.634} C_VEL
LIN {X 0,Y 273.916,Z 270.697,A -85,B 0,C 180,E1 -19440.674,E2 -19440.674} C_VEL
LIN {X 0,Y 273.368,Z 269.615,A -85,B 0,C 180,E1 -19441.2,E2 -19441.2} C_VEL
LIN {X 0,Y 270.914,Z 266.995,A -85,B 0,C 180,E1 -19443.576,E2 -19443.576} C_VEL
LIN {X 0,Y 269.946,Z 265.048,A -85,B 0,C 180,E1 -19444.853,E2 -19444.853} C_VEL
LIN {X 0,Y 266.907,Z 262.61,A -85,B 0,C 180,E1 -19450.621,E2 -19450.621} C_VEL
LIN {X 0,Y 266.587,Z 262.106,A -85,B 0,C 180,E1 -19453.724,E2 -19453.724} C_VEL
LIN {X 0,Y 267.867,Z 263.923,A -85,B 0,C 180,E1 -19458.747,E2 -19458.747} C_VEL
LIN {X 0,Y 269.608,Z 265.132,A -85,B 0,C 180,E1 -19461.403,E2 -19461.403} C_VEL
LIN {X 0,Y 271.529,Z 268.512,A -85,B 0,C 180,E1 -19463.802,E2 -19463.802} C_VEL
LIN {X 0,Y 273.409,Z 270.371,A -85,B 0,C 180,E1 -19465.543,E2 -19465.543} C_VEL
LIN {X 0,Y 276.109,Z 274.249,A -85,B 0,C 180,E1 -19467.761,E2 -19467.761} C_VEL
LIN {X 0,Y 277.321,Z 275.896,A -85,B 0,C 180,E1 -19468.622,E2 -19468.622} C_VEL
LIN {X 0,Y 280.982,Z 281.543,A -85,B 0,C 180,E1 -19471.01,E2 -19471.01} C_VEL
LIN {X 0,Y 284.744,Z 287.801,A -85,B 0,C 180,E1 -19473.134,E2 -19473.134} C_VEL
LIN {X 0,Y 289.73,Z 296.913,A -85,B 0,C 180,E1 -19475.636,E2 -19475.636} C_VEL
LIN {X 0,Y 294.857,Z 307.189,A -85,B 0,C 180,E1 -19477.918,E2 -19477.918} C_VEL
LIN {X 0,Y 299.414,Z 317.475,A -85,B 0,C 180,E1 -19479.79,E2 -19479.79} C_VEL
LIN {X 0,Y 290.867,Z 432.084,A -85,B 0,C 180,E1 -19482.62,E2 -19482.62} C_VEL
LIN {X 0,Y 288.477,Z 449.289,A -85,B 0,C 180,E1 -19483.229,E2 -19483.229} C_VEL
LIN {X 0,Y 285.393,Z 465.501,A -85,B 0,C 180,E1 -19484.045,E2 -19484.045} C_VEL
LIN {X 0,Y 281.479,Z 481.844,A -85,B 0,C 180,E1 -19485.14,E2 -19485.14} C_VEL
LIN {X 0,Y 277.517,Z 496.025,A -85,B 0,C 180,E1 -19486.36,E2 -19486.36} C_VEL
LIN {X 0,Y 272.705,Z 510.764,A -85,B 0,C 180,E1 -19487.926,E2 -19487.926} C_VEL
LIN {X 0,Y 267.825,Z 523.998,A -85,B 0,C 180,E1 -19489.677,E2 -19489.677} C_VEL
LIN {X 0,Y 263.058,Z 535.959,A -85,B 0,C 180,E1 -19491.596,E2 -19491.596} C_VEL
LIN {X 0,Y 258.311,Z 547.006,A -85,B 0,C 180,E1 -19493.715,E2 -19493.715} C_VEL
LIN {X 0,Y 252.948,Z 558.749,A -85,B 0,C 180,E1 -19496.462,E2 -19496.462} C_VEL
LIN {X 0,Y 248.18,Z 568.845,A -85,B 0,C 180,E1 -19499.351,E2 -19499.351} C_VEL
LIN {X 0,Y 243.837,Z 577.959,A -85,B 0,C 180,E1 -19502.535,E2 -19502.535} C_VEL
LIN {X 0,Y 240.313,Z 585.619,A -85,B 0,C 180,E1 -19505.827,E2 -19505.827} C_VEL
LIN {X 0,Y 236.888,Z 593.385,A -85,B 0,C 180,E1 -19510.048,E2 -19510.048} C_VEL
LIN {X 0,Y 234.591,Z 599.351,A -85,B 0,C 180,E1 -19514.354,E2 -19514.354} C_VEL
LIN {X 0,Y 233.343,Z 602.902,A -85,B 0,C 180,E1 -19517.825,E2 -19517.825} C_VEL
LIN {X 0,Y 232.813,Z 605.508,A -85,B 0,C 180,E1 -19521.315,E2 -19521.315} C_VEL
LIN {X 0,Y 232.646,Z 607.261,A -85,B 0,C 180,E1 -19525.475,E2 -19525.475} C_VEL
LIN {X 0,Y 232.741,Z 607.703,A -85,B 0,C 180,E1 -19528.265,E2 -19528.265} C_VEL
LIN {X 0,Y 232.821,Z 607.609,A -85,B 0,C 180,E1 -19529.996,E2 -19529.996} C_VEL
LIN {X 0,Y 232.683,Z 606.741,A -85,B 0,C 180,E1 -19533.459,E2 -19533.459} C_VEL
LIN {X 0,Y 232.726,Z 605.942,A -85,B 0,C 180,E1 -19535.193,E2 -19535.193} C_VEL
LIN {X 0,Y 232.805,Z 603.488,A -85,B 0,C 180,E1 -19538.677,E2 -19538.677} C_VEL
LIN {X 0,Y 233.311,Z 600.061,A -85,B 0,C 180,E1 -19542.168,E2 -19542.168} C_VEL
LIN {X 0,Y 234.458,Z 595.429,A -85,B 0,C 180,E1 -19545.646,E2 -19545.646} C_VEL
LIN {X 0,Y 236.068,Z 589.65,A -85,B 0,C 180,E1 -19549.111,E2 -19549.111} C_VEL
LIN {X 0,Y 238.408,Z 582.598,A -85,B 0,C 180,E1 -19552.528,E2 -19552.528} C_VEL
LIN {X 0,Y 241.818,Z 572.864,A -85,B 0,C 180,E1 -19556.303,E2 -19556.303} C_VEL
LIN {X 0,Y 245.728,Z 562.382,A -85,B 0,C 180,E1 -19559.556,E2 -19559.556} C_VEL
LIN {X 0,Y 249.744,Z 551.165,A -85,B 0,C 180,E1 -19562.412,E2 -19562.412} C_VEL
LIN {X 0,Y 254.138,Z 538.713,A -85,B 0,C 180,E1 -19565.011,E2 -19565.011} C_VEL
LIN {X 0,Y 258.487,Z 525.805,A -85,B 0,C 180,E1 -19567.219,E2 -19567.219} C_VEL
LIN {X 0,Y 262.295,Z 513.251,A -85,B 0,C 180,E1 -19569.011,E2 -19569.011} C_VEL
LIN {X 0,Y 266.063,Z 499.802,A -85,B 0,C 180,E1 -19570.57,E2 -19570.57} C_VEL
LIN {X 0,Y 269.731,Z 484.679,A -85,B 0,C 180,E1 -19572.006,E2 -19572.006} C_VEL
LIN {X 0,Y 272.865,Z 469.368,A -85,B 0,C 180,E1 -19573.162,E2 -19573.162} C_VEL
LIN {X 0,Y 275.681,Z 452.963,A -85,B 0,C 180,E1 -19574.082,E2 -19574.082} C_VEL
LIN {X 0,Y 277.815,Z 435.541,A -85,B 0,C 180,E1 -19574.774,E2 -19574.774} C_VEL
LIN {X 0,Y 279.887,Z 402.582,A -85,B 0,C 180,E1 -19575.656,E2 -19575.656} C_VEL
LIN {X 0,Y 285.466,Z 311.484,A -85,B 0,C 180,E1 -19577.903,E2 -19577.903} C_VEL
LIN {X 0,Y 279.602,Z 298.816,A -85,B 0,C 180,E1 -19579.53,E2 -19579.53} C_VEL
LIN {X 0,Y 272.468,Z 285.007,A -85,B 0,C 180,E1 -19581.577,E2 -19581.577} C_VEL
LIN {X 0,Y 264.948,Z 271.572,A -85,B 0,C 180,E1 -19583.888,E2 -19583.888} C_VEL
LIN {X 0,Y 258.367,Z 260.814,A -85,B 0,C 180,E1 -19586.043,E2 -19586.043} C_VEL
LIN {X 0,Y 254.527,Z 254.874,A -85,B 0,C 180,E1 -19587.373,E2 -19587.373} C_VEL
LIN {X 0,Y 249.435,Z 248.087,A -85,B 0,C 180,E1 -19589.187,E2 -19589.187} C_VEL
LIN {X 0,Y 246.064,Z 243.641,A -85,B 0,C 180,E1 -19590.469,E2 -19590.469} C_VEL
LIN {X 0,Y 243.493,Z 240.358,A -85,B 0,C 180,E1 -19591.476,E2 -19591.476} C_VEL
LIN {X 0,Y 242.492,Z 238.926,A -85,B 0,C 180,E1 -19591.886,E2 -19591.886} C_VEL
LIN {X 0,Y 240.008,Z 236.184,A -85,B 0,C 180,E1 -19592.89,E2 -19592.89} C_VEL
LIN {X 0,Y 238.793,Z 233.951,A -85,B 0,C 180,E1 -19593.45,E2 -19593.45} C_VEL
LIN {X 0,Y 236.337,Z 231.865,A -85,B 0,C 180,E1 -19594.481,E2 -19594.481} C_VEL
LIN {X 0,Y 235.174,Z 229.531,A -85,B 0,C 180,E1 -19595.069,E2 -19595.069} C_VEL
LIN {X 0,Y 234.986,Z 228.505,A -85,B 0,C 180,E1 -19595.248,E2 -19595.248} C_VEL
LIN {X 0,Y 235.019,Z 228.489,A -85,B 0,C 180,E1 -19598.971,E2 -19598.971} C_VEL
LIN {X 0,Y 235.092,Z 228.507,A -85,B 0,C 180,E1 -19603.042,E2 -19603.042} C_VEL
LIN {X 0,Y 235.091,Z 228.462,A -85,B 0,C 180,E1 -19607.922,E2 -19607.922} C_VEL
LIN {X 0,Y 235.35,Z 228.48,A -85,B 0,C 180,E1 -19611.414,E2 -19611.414} C_VEL
LIN {X 0,Y 235.376,Z 228.464,A -85,B 0,C 180,E1 -19613.141,E2 -19613.141} C_VEL
LIN {X 0,Y 235.568,Z 228.412,A -85,B 0,C 180,E1 -19618.291,E2 -19618.291} C_VEL
LIN {X 0,Y 235.568,Z 228.451,A -85,B 0,C 180,E1 -19621.711,E2 -19621.711} C_VEL
LIN {X 0,Y 235.347,Z 228.47,A -85,B 0,C 180,E1 -19626.861,E2 -19626.861} C_VEL
LIN {X 0,Y 235.188,Z 228.473,A -85,B 0,C 180,E1 -19630.33,E2 -19630.33} C_VEL
LIN {X 0,Y 235.088,Z 228.511,A -85,B 0,C 180,E1 -19635.609,E2 -19635.609} C_VEL
LIN {X 0,Y 234.985,Z 228.491,A -85,B 0,C 180,E1 -19639.209,E2 -19639.209} C_VEL
LIN {X 0,Y 234.939,Z 228.53,A -85,B 0,C 180,E1 -19642.886,E2 -19642.886} C_VEL
LIN {X 0,Y 234.949,Z 228.499,A -85,B 0,C 180,E1 -19646.661,E2 -19646.661} C_VEL
LIN {X 0,Y 234.912,Z 228.528,A -85,B 0,C 180,E1 -19650.572,E2 -19650.572} C_VEL
LIN {X 0,Y 234.912,Z 228.519,A -85,B 0,C 180,E1 -19654.642,E2 -19654.642} C_VEL
LIN {X 0,Y 234.897,Z 228.51,A -85,B 0,C 180,E1 -19658.94,E2 -19658.94} C_VEL
LIN {X 0,Y 234.863,Z 228.529,A -85,B 0,C 180,E1 -19663.493,E2 -19663.493} C_VEL
LIN {X 0,Y 234.865,Z 228.525,A -85,B 0,C 180,E1 -19666.517,E2 -19666.517} C_VEL
LIN {X 0,Y 234.906,Z 228.516,A -85,B 0,C 180,E1 -19671.083,E2 -19671.083} C_VEL
LIN {X 0,Y 234.964,Z 228.659,A -85,B 0,C 180,E1 -19672.322,E2 -19672.322} C_VEL
LIN {X 0,Y 235.836,Z 231.221,A -85,B 0,C 180,E1 -19672.811,E2 -19672.811} C_VEL
LIN {X 0,Y 237.846,Z 233.427,A -85,B 0,C 180,E1 -19673.686,E2 -19673.686} C_VEL
LIN {X 0,Y 239.022,Z 234.227,A -85,B 0,C 180,E1 -19674.157,E2 -19674.157} C_VEL
LIN {X 0,Y 240.923,Z 237.417,A -85,B 0,C 180,E1 -19675.009,E2 -19675.009} C_VEL
LIN {X 0,Y 243.061,Z 239.648,A -85,B 0,C 180,E1 -19675.866,E2 -19675.866} C_VEL
LIN {X 0,Y 245.55,Z 243.145,A -85,B 0,C 180,E1 -19676.871,E2 -19676.871} C_VEL
LIN {X 0,Y 247.133,Z 244.964,A -85,B 0,C 180,E1 -19677.467,E2 -19677.467} C_VEL
LIN {X 0,Y 251.253,Z 250.578,A -85,B 0,C 180,E1 -19679.001,E2 -19679.001} C_VEL
LIN {X 0,Y 256.708,Z 257.883,A -85,B 0,C 180,E1 -19680.899,E2 -19680.899} C_VEL
LIN {X 0,Y 265.203,Z 270.253,A -85,B 0,C 180,E1 -19683.634,E2 -19683.634} C_VEL
LIN {X 0,Y 272.67,Z 281.96,A -85,B 0,C 180,E1 -19685.859,E2 -19685.859} C_VEL
LIN {X 0,Y 280.548,Z 295.166,A -85,B 0,C 180,E1 -19688.037,E2 -19688.037} C_VEL
LIN {X 0,Y 285.52,Z 304.233,A -85,B 0,C 180,E1 -19689.355,E2 -19689.355} C_VEL
LIN {X 0,Y 278.477,Z 420.438,A -85,B 0,C 180,E1 -19692.281,E2 -19692.281} C_VEL
LIN {X 0,Y 276.685,Z 436.987,A -85,B 0,C 180,E1 -19692.925,E2 -19692.925} C_VEL
LIN {X 0,Y 274.228,Z 453.352,A -85,B 0,C 180,E1 -19693.821,E2 -19693.821} C_VEL
LIN {X 0,Y 271.237,Z 469.317,A -85,B 0,C 180,E1 -19694.987,E2 -19694.987} C_VEL
LIN {X 0,Y 268.009,Z 484.018,A -85,B 0,C 180,E1 -19696.353,E2 -19696.353} C_VEL
LIN {X 0,Y 264.373,Z 497.776,A -85,B 0,C 180,E1 -19697.92,E2 -19697.92} C_VEL
LIN {X 0,Y 260.525,Z 510.755,A -85,B 0,C 180,E1 -19699.709,E2 -19699.709} C_VEL
LIN {X 0,Y 256.272,Z 524.003,A -85,B 0,C 180,E1 -19701.925,E2 -19701.925} C_VEL
LIN {X 0,Y 252.026,Z 536.243,A -85,B 0,C 180,E1 -19704.403,E2 -19704.403} C_VEL
LIN {X 0,Y 247.958,Z 547.407,A -85,B 0,C 180,E1 -19707.161,E2 -19707.161} C_VEL
LIN {X 0,Y 244.358,Z 556.934,A -85,B 0,C 180,E1 -19710.004,E2 -19710.004} C_VEL
LIN {X 0,Y 240.829,Z 566.2,A -85,B 0,C 180,E1 -19713.35,E2 -19713.35} C_VEL
LIN {X 0,Y 238.038,Z 573.922,A -85,B 0,C 180,E1 -19716.786,E2 -19716.786} C_VEL
LIN {X 0,Y 235.847,Z 580.516,A -85,B 0,C 180,E1 -19720.459,E2 -19720.459} C_VEL
LIN {X 0,Y 234.359,Z 585.324,A -85,B 0,C 180,E1 -19723.885,E2 -19723.885} C_VEL
LIN {X 0,Y 233.245,Z 589.296,A -85,B 0,C 180,E1 -19727.54,E2 -19727.54} C_VEL
LIN {X 0,Y 232.532,Z 592.117,A -85,B 0,C 180,E1 -19731.269,E2 -19731.269} C_VEL
LIN {X 0,Y 232.25,Z 593.792,A -85,B 0,C 180,E1 -19735.069,E2 -19735.069} C_VEL
LIN {X 0,Y 232.336,Z 594.36,A -85,B 0,C 180,E1 -19738.95,E2 -19738.95} C_VEL
LIN {X 0,Y 232.636,Z 593.693,A -85,B 0,C 180,E1 -19742.945,E2 -19742.945} C_VEL
LIN {X 0,Y 233.116,Z 592.612,A -85,B 0,C 180,E1 -19745.51,E2 -19745.51} C_VEL
LIN {X 0,Y 234.158,Z 590.159,A -85,B 0,C 180,E1 -19749.075,E2 -19749.075} C_VEL
LIN {X 0,Y 236.032,Z 585.993,A -85,B 0,C 180,E1 -19753.226,E2 -19753.226} C_VEL
LIN {X 0,Y 237.984,Z 581.83,A -85,B 0,C 180,E1 -19756.349,E2 -19756.349} C_VEL
LIN {X 0,Y 241.098,Z 575.399,A -85,B 0,C 180,E1 -19760.11,E2 -19760.11} C_VEL
LIN {X 0,Y 244.846,Z 568.083,A -85,B 0,C 180,E1 -19763.489,E2 -19763.489} C_VEL
LIN {X 0,Y 248.772,Z 560.271,A -85,B 0,C 180,E1 -19766.453,E2 -19766.453} C_VEL
LIN {X 0,Y 253.293,Z 550.93,A -85,B 0,C 180,E1 -19769.336,E2 -19769.336} C_VEL
LIN {X 0,Y 258.416,Z 540.008,A -85,B 0,C 180,E1 -19772.102,E2 -19772.102} C_VEL
LIN {X 0,Y 263.722,Z 527.84,A -85,B 0,C 180,E1 -19774.632,E2 -19774.632} C_VEL
LIN {X 0,Y 268.884,Z 515.138,A -85,B 0,C 180,E1 -19776.779,E2 -19776.779} C_VEL
LIN {X 0,Y 274.155,Z 500.633,A -85,B 0,C 180,E1 -19778.769,E2 -19778.769} C_VEL
LIN {X 0,Y 278.722,Z 486.138,A -85,B 0,C 180,E1 -19780.371,E2 -19780.371} C_VEL
LIN {X 0,Y 282.723,Z 471.434,A -85,B 0,C 180,E1 -19781.676,E2 -19781.676} C_VEL
LIN {X 0,Y 286.335,Z 455.435,A -85,B 0,C 180,E1 -19782.799,E2 -19782.799} C_VEL
LIN {X 0,Y 289.116,Z 439.942,A -85,B 0,C 180,E1 -19783.628,E2 -19783.628} C_VEL
LIN {X 0,Y 291.293,Z 423.609,A -85,B 0,C 180,E1 -19784.251,E2 -19784.251} C_VEL
LIN {X 0,Y 297.523,Z 340.757,A -85,B 0,C 180,E1 -19786.317,E2 -19786.317} C_VEL
LIN {X 0,Y 298.706,Z 325.325,A -85,B 0,C 180,E1 -19786.684,E2 -19786.684} C_VEL
LIN {X 0,Y 298.587,Z 322.257,A -85,B 0,C 180,E1 -19786.86,E2 -19786.86} C_VEL
LIN {X 0,Y 297.538,Z 318.563,A -85,B 0,C 180,E1 -19787.341,E2 -19787.341} C_VEL
LIN {X 0,Y 292.739,Z 309.8,A -85,B 0,C 180,E1 -19789.263,E2 -19789.263} C_VEL
LIN {X 0,Y 288.796,Z 302.679,A -85,B 0,C 180,E1 -19791.017,E2 -19791.017} C_VEL
LIN {X 0,Y 284.481,Z 295.561,A -85,B 0,C 180,E1 -19793.12,E2 -19793.12} C_VEL
LIN {X 0,Y 280.257,Z 288.855,A -85,B 0,C 180,E1 -19795.454,E2 -19795.454} C_VEL
LIN {X 0,Y 277.641,Z 284.914,A -85,B 0,C 180,E1 -19797.097,E2 -19797.097} C_VEL
LIN {X 0,Y 274.62,Z 280.639,A -85,B 0,C 180,E1 -19799.243,E2 -19799.243} C_VEL
LIN {X 0,Y 272.169,Z 276.839,A -85,B 0,C 180,E1 -19801.342,E2 -19801.342} C_VEL
LIN {X 0,Y 269.183,Z 272.943,A -85,B 0,C 180,E1 -19804.492,E2 -19804.492} C_VEL
LIN {X 0,Y 268.656,Z 271.907,A -85,B 0,C 180,E1 -19805.253,E2 -19805.253} C_VEL
LIN {X 0,Y 265.937,Z 269.647,A -85,B 0,C 180,E1 -19810.66,E2 -19810.66} C_VEL
LIN {X 0,Y 265.636,Z 269.143,A -85,B 0,C 180,E1 -19813.775,E2 -19813.775} C_VEL
LIN {X 0,Y 267.623,Z 271.468,A -85,B 0,C 180,E1 -19819.961,E2 -19819.961} C_VEL
LIN {X 0,Y 268.413,Z 272.044,A -85,B 0,C 180,E1 -19821.11,E2 -19821.11} C_VEL
LIN {X 0,Y 270.256,Z 275.348,A -85,B 0,C 180,E1 -19823.514,E2 -19823.514} C_VEL
LIN {X 0,Y 271.985,Z 277.108,A -85,B 0,C 180,E1 -19825.174,E2 -19825.174} C_VEL
LIN {X 0,Y 274.523,Z 280.878,A -85,B 0,C 180,E1 -19827.348,E2 -19827.348} C_VEL
LIN {X 0,Y 275.797,Z 282.768,A -85,B 0,C 180,E1 -19828.308,E2 -19828.308} C_VEL
LIN {X 0,Y 279.005,Z 287.847,A -85,B 0,C 180,E1 -19830.475,E2 -19830.475} C_VEL
LIN {X 0,Y 282.608,Z 294.138,A -85,B 0,C 180,E1 -19832.616,E2 -19832.616} C_VEL
LIN {X 0,Y 287.283,Z 302.958,A -85,B 0,C 180,E1 -19835.07,E2 -19835.07} C_VEL
LIN {X 0,Y 292.162,Z 313.266,A -85,B 0,C 180,E1 -19837.356,E2 -19837.356} C_VEL
LIN {X 0,Y 295.297,Z 320.389,A -85,B 0,C 180,E1 -19838.701,E2 -19838.701} C_VEL
LIN {X 0,Y 286.577,Z 432.565,A -85,B 0,C 180,E1 -19841.501,E2 -19841.501} C_VEL
LIN {X 0,Y 284.031,Z 450.138,A -85,B 0,C 180,E1 -19842.135,E2 -19842.135} C_VEL
LIN {X 0,Y 280.859,Z 466.05,A -85,B 0,C 180,E1 -19842.949,E2 -19842.949} C_VEL
LIN {X 0,Y 277.101,Z 481.248,A -85,B 0,C 180,E1 -19843.971,E2 -19843.971} C_VEL
LIN {X 0,Y 272.994,Z 495.48,A -85,B 0,C 180,E1 -19845.188,E2 -19845.188} C_VEL
LIN {X 0,Y 268.014,Z 510.198,A -85,B 0,C 180,E1 -19846.757,E2 -19846.757} C_VEL
LIN {X 0,Y 263.059,Z 523.147,A -85,B 0,C 180,E1 -19848.468,E2 -19848.468} C_VEL
LIN {X 0,Y 257.538,Z 536.437,A -85,B 0,C 180,E1 -19850.616,E2 -19850.616} C_VEL
LIN {X 0,Y 251.851,Z 549.056,A -85,B 0,C 180,E1 -19853.129,E2 -19853.129} C_VEL
LIN {X 0,Y 246.833,Z 559.481,A -85,B 0,C 180,E1 -19855.659,E2 -19855.659} C_VEL
LIN {X 0,Y 242.057,Z 569.029,A -85,B 0,C 180,E1 -19858.488,E2 -19858.488} C_VEL
LIN {X 0,Y 237.502,Z 578.068,A -85,B 0,C 180,E1 -19861.737,E2 -19861.737} C_VEL
LIN {X 0,Y 233.754,Z 585.696,A -85,B 0,C 180,E1 -19865.104,E2 -19865.104} C_VEL
LIN {X 0,Y 230.118,Z 593.385,A -85,B 0,C 180,E1 -19869.434,E2 -19869.434} C_VEL
LIN {X 0,Y 227.685,Z 599.293,A -85,B 0,C 180,E1 -19873.867,E2 -19873.867} C_VEL
LIN {X 0,Y 226.34,Z 602.796,A -85,B 0,C 180,E1 -19877.442,E2 -19877.442} C_VEL
LIN {X 0,Y 225.735,Z 605.378,A -85,B 0,C 180,E1 -19881.04,E2 -19881.04} C_VEL
LIN {X 0,Y 225.552,Z 607.17,A -85,B 0,C 180,E1 -19885.618,E2 -19885.618} C_VEL
LIN {X 0,Y 225.654,Z 607.507,A -85,B 0,C 180,E1 -19888.211,E2 -19888.211} C_VEL
LIN {X 0,Y 225.732,Z 607.392,A -85,B 0,C 180,E1 -19889.996,E2 -19889.996} C_VEL
LIN {X 0,Y 225.596,Z 606.483,A -85,B 0,C 180,E1 -19893.568,E2 -19893.568} C_VEL
LIN {X 0,Y 225.631,Z 605.679,A -85,B 0,C 180,E1 -19895.357,E2 -19895.357} C_VEL
LIN {X 0,Y 225.725,Z 603.184,A -85,B 0,C 180,E1 -19898.951,E2 -19898.951} C_VEL
LIN {X 0,Y 226.314,Z 599.71,A -85,B 0,C 180,E1 -19902.55,E2 -19902.55} C_VEL
LIN {X 0,Y 227.533,Z 595.047,A -85,B 0,C 180,E1 -19906.135,E2 -19906.135} C_VEL
LIN {X 0,Y 229.255,Z 589.208,A -85,B 0,C 180,E1 -19909.702,E2 -19909.702} C_VEL
LIN {X 0,Y 231.754,Z 582.108,A -85,B 0,C 180,E1 -19913.212,E2 -19913.212} C_VEL
LIN {X 0,Y 235.346,Z 572.295,A -85,B 0,C 180,E1 -19917.085,E2 -19917.085} C_VEL
LIN {X 0,Y 239.45,Z 561.744,A -85,B 0,C 180,E1 -19920.411,E2 -19920.411} C_VEL
LIN {X 0,Y 243.517,Z 550.774,A -85,B 0,C 180,E1 -19923.247,E2 -19923.247} C_VEL
LIN {X 0,Y 247.552,Z 539.874,A -85,B 0,C 180,E1 -19925.585,E2 -19925.585} C_VEL
LIN {X 0,Y 251.984,Z 527.233,A -85,B 0,C 180,E1 -19927.843,E2 -19927.843} C_VEL
LIN {X 0,Y 256.324,Z 513.495,A -85,B 0,C 180,E1 -19929.852,E2 -19929.852} C_VEL
LIN {X 0,Y 260.193,Z 500.189,A -85,B 0,C 180,E1 -19931.428,E2 -19931.428} C_VEL
LIN {X 0,Y 263.955,Z 485.208,A -85,B 0,C 180,E1 -19932.885,E2 -19932.885} C_VEL
LIN {X 0,Y 267.185,Z 470.115,A -85,B 0,C 180,E1 -19934.053,E2 -19934.053} C_VEL
LIN {X 0,Y 270.128,Z 453.462,A -85,B 0,C 180,E1 -19935.006,E2 -19935.006} C_VEL
LIN {X 0,Y 272.212,Z 437.232,A -85,B 0,C 180,E1 -19935.676,E2 -19935.676} C_VEL
LIN {X 0,Y 273.871,Z 414.414,A -85,B 0,C 180,E1 -19936.323,E2 -19936.323} C_VEL
LIN {X 0,Y 280.143,Z 313.645,A -85,B 0,C 180,E1 -19938.86,E2 -19938.86} C_VEL
LIN {X 0,Y 273.326,Z 299.27,A -85,B 0,C 180,E1 -19940.82,E2 -19940.82} C_VEL
LIN {X 0,Y 266.249,Z 285.698,A -85,B 0,C 180,E1 -19942.976,E2 -19942.976} C_VEL
LIN {X 0,Y 258.394,Z 271.801,A -85,B 0,C 180,E1 -19945.531,E2 -19945.531} C_VEL
LIN {X 0,Y 251.781,Z 261.231,A -85,B 0,C 180,E1 -19947.845,E2 -19947.845} C_VEL
LIN {X 0,Y 245.845,Z 253.218,A -85,B 0,C 180,E1 -19950.035,E2 -19950.035} C_VEL
LIN {X 0,Y 242.778,Z 249.155,A -85,B 0,C 180,E1 -19951.237,E2 -19951.237} C_VEL
LIN {X 0,Y 239.422,Z 244.752,A -85,B 0,C 180,E1 -19952.612,E2 -19952.612} C_VEL
LIN {X 0,Y 236.836,Z 241.521,A -85,B 0,C 180,E1 -19953.722,E2 -19953.722} C_VEL
LIN {X 0,Y 235.763,Z 239.959,A -85,B 0,C 180,E1 -19954.213,E2 -19954.213} C_VEL
LIN {X 0,Y 233.155,Z 237.098,A -85,B 0,C 180,E1 -19955.396,E2 -19955.396} C_VEL
LIN {X 0,Y 232.029,Z 234.985,A -85,B 0,C 180,E1 -19955.984,E2 -19955.984} C_VEL
LIN {X 0,Y 229.534,Z 233.092,A -85,B 0,C 180,E1 -19957.122,E2 -19957.122} C_VEL
LIN {X 0,Y 228.302,Z 230.791,A -85,B 0,C 180,E1 -19957.794,E2 -19957.794} C_VEL
LIN {X 0,Y 227.994,Z 229.377,A -85,B 0,C 180,E1 -19958.065,E2 -19958.065} C_VEL
LIN {X 0,Y 228.02,Z 229.38,A -85,B 0,C 180,E1 -19962.817,E2 -19962.817} C_VEL
LIN {X 0,Y 228.048,Z 229.339,A -85,B 0,C 180,E1 -19967.543,E2 -19967.543} C_VEL
LIN {X 0,Y 228.28,Z 229.357,A -85,B 0,C 180,E1 -19971.146,E2 -19971.146} C_VEL
LIN {X 0,Y 228.327,Z 229.346,A -85,B 0,C 180,E1 -19972.929,E2 -19972.929} C_VEL
LIN {X 0,Y 228.527,Z 229.287,A -85,B 0,C 180,E1 -19978.239,E2 -19978.239} C_VEL
LIN {X 0,Y 228.527,Z 229.327,A -85,B 0,C 180,E1 -19981.763,E2 -19981.763} C_VEL
LIN {X 0,Y 228.298,Z 229.351,A -85,B 0,C 180,E1 -19987.074,E2 -19987.074} C_VEL
LIN {X 0,Y 228.119,Z 229.349,A -85,B 0,C 180,E1 -19990.653,E2 -19990.653} C_VEL
LIN {X 0,Y 228.033,Z 229.385,A -85,B 0,C 180,E1 -19996.105,E2 -19996.105} C_VEL
LIN {X 0,Y 227.919,Z 229.374,A -85,B 0,C 180,E1 -19999.829,E2 -19999.829} C_VEL
LIN {X 0,Y 227.892,Z 229.399,A -85,B 0,C 180,E1 -20003.636,E2 -20003.636} C_VEL
LIN {X 0,Y 227.866,Z 229.39,A -85,B 0,C 180,E1 -20007.559,E2 -20007.559} C_VEL
LIN {X 0,Y 227.851,Z 229.39,A -85,B 0,C 180,E1 -20011.626,E2 -20011.626} C_VEL
LIN {X 0,Y 227.864,Z 229.414,A -85,B 0,C 180,E1 -20015.876,E2 -20015.876} C_VEL
LIN {X 0,Y 227.795,Z 229.399,A -85,B 0,C 180,E1 -20020.385,E2 -20020.385} C_VEL
LIN {X 0,Y 227.812,Z 229.395,A -85,B 0,C 180,E1 -20025.2,E2 -20025.2} C_VEL
LIN {X 0,Y 227.821,Z 229.519,A -85,B 0,C 180,E1 -20029.429,E2 -20029.429} C_VEL
LIN {X 0,Y 228.594,Z 231.894,A -85,B 0,C 180,E1 -20029.92,E2 -20029.92} C_VEL
LIN {X 0,Y 230.631,Z 234.199,A -85,B 0,C 180,E1 -20030.93,E2 -20030.93} C_VEL
LIN {X 0,Y 232.18,Z 235.279,A -85,B 0,C 180,E1 -20031.634,E2 -20031.634} C_VEL
LIN {X 0,Y 233.934,Z 238.33,A -85,B 0,C 180,E1 -20032.514,E2 -20032.514} C_VEL
LIN {X 0,Y 236.375,Z 240.669,A -85,B 0,C 180,E1 -20033.572,E2 -20033.572} C_VEL
LIN {X 0,Y 238.822,Z 244.117,A -85,B 0,C 180,E1 -20034.653,E2 -20034.653} C_VEL
LIN {X 0,Y 240.323,Z 245.864,A -85,B 0,C 180,E1 -20035.275,E2 -20035.275} C_VEL
LIN {X 0,Y 243.324,Z 249.754,A -85,B 0,C 180,E1 -20036.5,E2 -20036.5} C_VEL
LIN {X 0,Y 251.198,Z 260.396,A -85,B 0,C 180,E1 -20039.469,E2 -20039.469} C_VEL
LIN {X 0,Y 259.181,Z 271.928,A -85,B 0,C 180,E1 -20042.2,E2 -20042.2} C_VEL
LIN {X 0,Y 268.156,Z 285.917,A -85,B 0,C 180,E1 -20044.997,E2 -20044.997} C_VEL
LIN {X 0,Y 276.398,Z 299.92,A -85,B 0,C 180,E1 -20047.369,E2 -20047.369} C_VEL
LIN {X 0,Y 280.236,Z 306.966,A -85,B 0,C 180,E1 -20048.419,E2 -20048.419} C_VEL
LIN {X 0,Y 273.065,Z 421.228,A -85,B 0,C 180,E1 -20051.335,E2 -20051.335} C_VEL
LIN {X 0,Y 271.081,Z 438.488,A -85,B 0,C 180,E1 -20052.025,E2 -20052.025} C_VEL
LIN {X 0,Y 268.682,Z 453.817,A -85,B 0,C 180,E1 -20052.891,E2 -20052.891} C_VEL
LIN {X 0,Y 265.612,Z 469.71,A -85,B 0,C 180,E1 -20054.071,E2 -20054.071} C_VEL
LIN {X 0,Y 262.274,Z 484.377,A -85,B 0,C 180,E1 -20055.455,E2 -20055.455} C_VEL
LIN {X 0,Y 258.522,Z 498.12,A -85,B 0,C 180,E1 -20057.044,E2 -20057.044} C_VEL
LIN {X 0,Y 254.545,Z 511.079,A -85,B 0,C 180,E1 -20058.861,E2 -20058.861} C_VEL
LIN {X 0,Y 250.15,Z 524.307,A -85,B 0,C 180,E1 -20061.115,E2 -20061.115} C_VEL
LIN {X 0,Y 246.061,Z 535.674,A -85,B 0,C 180,E1 -20063.444,E2 -20063.444} C_VEL
LIN {X 0,Y 241.807,Z 546.933,A -85,B 0,C 180,E1 -20066.255,E2 -20066.255} C_VEL
LIN {X 0,Y 238.009,Z 556.58,A -85,B 0,C 180,E1 -20069.158,E2 -20069.158} C_VEL
LIN {X 0,Y 234.322,Z 565.939,A -85,B 0,C 180,E1 -20072.583,E2 -20072.583} C_VEL
LIN {X 0,Y 231.35,Z 573.761,A -85,B 0,C 180,E1 -20076.107,E2 -20076.107} C_VEL
LIN {X 0,Y 229.12,Z 579.998,A -85,B 0,C 180,E1 -20079.634,E2 -20079.634} C_VEL
LIN {X 0,Y 227.431,Z 585.287,A -85,B 0,C 180,E1 -20083.405,E2 -20083.405} C_VEL
LIN {X 0,Y 226.475,Z 588.408,A -85,B 0,C 180,E1 -20086.222,E2 -20086.222} C_VEL
LIN {X 0,Y 225.647,Z 591.569,A -85,B 0,C 180,E1 -20090.039,E2 -20090.039} C_VEL
LIN {X 0,Y 225.19,Z 593.651,A -85,B 0,C 180,E1 -20093.94,E2 -20093.94} C_VEL
LIN {X 0,Y 225.19,Z 594.508,A -85,B 0,C 180,E1 -20097.917,E2 -20097.917} C_VEL
LIN {X 0,Y 225.476,Z 594.212,A -85,B 0,C 180,E1 -20102.001,E2 -20102.001} C_VEL
LIN {X 0,Y 226.175,Z 592.66,A -85,B 0,C 180,E1 -20106.189,E2 -20106.189} C_VEL
LIN {X 0,Y 227.568,Z 589.7,A -85,B 0,C 180,E1 -20110.436,E2 -20110.436} C_VEL
LIN {X 0,Y 229.752,Z 585.201,A -85,B 0,C 180,E1 -20114.717,E2 -20114.717} C_VEL
LIN {X 0,Y 232.267,Z 580.22,A -85,B 0,C 180,E1 -20118.264,E2 -20118.264} C_VEL
LIN {X 0,Y 235.954,Z 573.286,A -85,B 0,C 180,E1 -20122.125,E2 -20122.125} C_VEL
LIN {X 0,Y 239.682,Z 566.374,A -85,B 0,C 180,E1 -20125.191,E2 -20125.191} C_VEL
LIN {X 0,Y 244.554,Z 557.004,A -85,B 0,C 180,E1 -20128.569,E2 -20128.569} C_VEL
LIN {X 0,Y 249.96,Z 546.348,A -85,B 0,C 180,E1 -20131.654,E2 -20131.654} C_VEL
LIN {X 0,Y 255.725,Z 534.256,A -85,B 0,C 180,E1 -20134.473,E2 -20134.473} C_VEL
LIN {X 0,Y 261.018,Z 522.224,A -85,B 0,C 180,E1 -20136.76,E2 -20136.76} C_VEL
LIN {X 0,Y 266.529,Z 508.516,A -85,B 0,C 180,E1 -20138.878,E2 -20138.878} C_VEL
LIN {X 0,Y 271.965,Z 493.075,A -85,B 0,C 180,E1 -20140.797,E2 -20140.797} C_VEL
LIN {X 0,Y 276.435,Z 478.411,A -85,B 0,C 180,E1 -20142.236,E2 -20142.236} C_VEL
LIN {X 0,Y 280.207,Z 463.575,A -85,B 0,C 180,E1 -20143.409,E2 -20143.409} C_VEL
LIN {X 0,Y 283.493,Z 447.844,A -85,B 0,C 180,E1 -20144.374,E2 -20144.374} C_VEL
LIN {X 0,Y 286.07,Z 431.7,A -85,B 0,C 180,E1 -20145.114,E2 -20145.114} C_VEL
LIN {X 0,Y 287.985,Z 413.969,A -85,B 0,C 180,E1 -20145.654,E2 -20145.654} C_VEL
LIN {X 0,Y 295.59,Z 315.228,A -85,B 0,C 180,E1 -20148.09,E2 -20148.09} C_VEL
LIN {X 0,Y 292.739,Z 309.8,A -85,B 0,C 180,E1 -20149.263,E2 -20149.263} C_VEL
LIN {X 0,Y 291.458,Z 307.43,A -85,B 0,C 180,E1 -20149.816,E2 -20149.816} C_VEL
LIN {X 0,Y 289.126,Z 304.983,A -85,B 0,C 180,E1 -20150.77,E2 -20150.77} C_VEL
LIN {X 0,Y 281.776,Z 300.398,A -85,B 0,C 180,E1 -20153.973,E2 -20153.973} C_VEL
LIN {X 0,Y 280.45,Z 298.758,A -85,B 0,C 180,E1 -20154.675,E2 -20154.675} C_VEL
LIN {X 0,Y 276.211,Z 291.791,A -85,B 0,C 180,E1 -20157.338,E2 -20157.338} C_VEL
LIN {X 0,Y 272.958,Z 287.182,A -85,B 0,C 180,E1 -20159.726,E2 -20159.726} C_VEL
LIN {X 0,Y 270.378,Z 283.086,A -85,B 0,C 180,E1 -20162.076,E2 -20162.076} C_VEL
LIN {X 0,Y 267.992,Z 279.886,A -85,B 0,C 180,E1 -20164.752,E2 -20164.752} C_VEL
LIN {X 0,Y 267.384,Z 278.752,A -85,B 0,C 180,E1 -20165.652,E2 -20165.652} C_VEL
LIN {X 0,Y 264.903,Z 276.609,A -85,B 0,C 180,E1 -20170.993,E2 -20170.993} C_VEL
LIN {X 0,Y 264.686,Z 276.177,A -85,B 0,C 180,E1 -20173.825,E2 -20173.825} C_VEL
LIN {X 0,Y 266.702,Z 278.529,A -85,B 0,C 180,E1 -20180.033,E2 -20180.033} C_VEL
LIN {X 0,Y 267.31,Z 279.147,A -85,B 0,C 180,E1 -20180.953,E2 -20180.953} C_VEL
LIN {X 0,Y 269.18,Z 282.409,A -85,B 0,C 180,E1 -20183.427,E2 -20183.427} C_VEL
LIN {X 0,Y 270.582,Z 283.949,A -85,B 0,C 180,E1 -20184.821,E2 -20184.821} C_VEL
LIN {X 0,Y 273.873,Z 288.884,A -85,B 0,C 180,E1 -20187.659,E2 -20187.659} C_VEL
LIN {X 0,Y 276.998,Z 294.081,A -85,B 0,C 180,E1 -20189.897,E2 -20189.897} C_VEL
LIN {X 0,Y 280.182,Z 299.825,A -85,B 0,C 180,E1 -20191.904,E2 -20191.904} C_VEL
LIN {X 0,Y 284.458,Z 308.229,A -85,B 0,C 180,E1 -20194.283,E2 -20194.283} C_VEL
LIN {X 0,Y 288.911,Z 317.874,A -85,B 0,C 180,E1 -20196.488,E2 -20196.488} C_VEL
LIN {X 0,Y 291.281,Z 323.484,A -85,B 0,C 180,E1 -20197.587,E2 -20197.587} C_VEL
LIN {X 0,Y 284.653,Z 406.949,A -85,B 0,C 180,E1 -20199.654,E2 -20199.654} C_VEL
LIN {X 0,Y 282.344,Z 433.764,A -85,B 0,C 180,E1 -20200.371,E2 -20200.371} C_VEL
LIN {X 0,Y 279.701,Z 451.066,A -85,B 0,C 180,E1 -20201.009,E2 -20201.009} C_VEL
LIN {X 0,Y 276.15,Z 467.9,A -85,B 0,C 180,E1 -20201.889,E2 -20201.889} C_VEL
LIN {X 0,Y 271.735,Z 484.525,A -85,B 0,C 180,E1 -20203.057,E2 -20203.057} C_VEL
LIN {X 0,Y 267.032,Z 499.609,A -85,B 0,C 180,E1 -20204.444,E2 -20204.444} C_VEL
LIN {X 0,Y 261.937,Z 513.622,A -85,B 0,C 180,E1 -20206.03,E2 -20206.03} C_VEL
LIN {X 0,Y 256.513,Z 527.079,A -85,B 0,C 180,E1 -20207.92,E2 -20207.92} C_VEL
LIN {X 0,Y 250.372,Z 540.789,A -85,B 0,C 180,E1 -20210.309,E2 -20210.309} C_VEL
LIN {X 0,Y 244.598,Z 552.663,A -85,B 0,C 180,E1 -20212.884,E2 -20212.884} C_VEL
LIN {X 0,Y 239.401,Z 562.843,A -85,B 0,C 180,E1 -20215.586,E2 -20215.586} C_VEL
LIN {X 0,Y 234.126,Z 572.798,A -85,B 0,C 180,E1 -20218.811,E2 -20218.811} C_VEL
LIN {X 0,Y 230.12,Z 580.221,A -85,B 0,C 180,E1 -20221.743,E2 -20221.743} C_VEL
LIN {X 0,Y 226.383,Z 587.385,A -85,B 0,C 180,E1 -20225.218,E2 -20225.218} C_VEL
LIN {X 0,Y 223.393,Z 593.383,A -85,B 0,C 180,E1 -20228.786,E2 -20228.786} C_VEL
LIN {X 0,Y 220.78,Z 599.244,A -85,B 0,C 180,E1 -20233.348,E2 -20233.348} C_VEL
LIN {X 0,Y 219.354,Z 602.694,A -85,B 0,C 180,E1 -20237.036,E2 -20237.036} C_VEL
LIN {X 0,Y 218.678,Z 605.238,A -85,B 0,C 180,E1 -20240.749,E2 -20240.749} C_VEL
LIN {X 0,Y 218.479,Z 607.048,A -85,B 0,C 180,E1 -20245.704,E2 -20245.704} C_VEL
LIN {X 0,Y 218.549,Z 607.301,A -85,B 0,C 180,E1 -20248.153,E2 -20248.153} C_VEL
LIN {X 0,Y 218.646,Z 607.174,A -85,B 0,C 180,E1 -20249.996,E2 -20249.996} C_VEL
LIN {X 0,Y 218.499,Z 606.217,A -85,B 0,C 180,E1 -20253.684,E2 -20253.684} C_VEL
LIN {X 0,Y 218.544,Z 605.398,A -85,B 0,C 180,E1 -20255.532,E2 -20255.532} C_VEL
LIN {X 0,Y 218.668,Z 602.867,A -85,B 0,C 180,E1 -20259.243,E2 -20259.243} C_VEL
LIN {X 0,Y 219.328,Z 599.341,A -85,B 0,C 180,E1 -20262.957,E2 -20262.957} C_VEL
LIN {X 0,Y 220.614,Z 594.648,A -85,B 0,C 180,E1 -20266.656,E2 -20266.656} C_VEL
LIN {X 0,Y 222.458,Z 588.749,A -85,B 0,C 180,E1 -20270.33,E2 -20270.33} C_VEL
LIN {X 0,Y 225.119,Z 581.588,A -85,B 0,C 180,E1 -20273.939,E2 -20273.939} C_VEL
LIN {X 0,Y 228.442,Z 572.893,A -85,B 0,C 180,E1 -20277.476,E2 -20277.476} C_VEL
LIN {X 0,Y 232.067,Z 563.875,A -85,B 0,C 180,E1 -20280.476,E2 -20280.476} C_VEL
LIN {X 0,Y 236.541,Z 552.588,A -85,B 0,C 180,E1 -20283.58,E2 -20283.58} C_VEL
LIN {X 0,Y 240.989,Z 541.035,A -85,B 0,C 180,E1 -20286.19,E2 -20286.19} C_VEL
LIN {X 0,Y 245.932,Z 527.464,A -85,B 0,C 180,E1 -20288.684,E2 -20288.684} C_VEL
LIN {X 0,Y 250.413,Z 513.734,A -85,B 0,C 180,E1 -20290.733,E2 -20290.733} C_VEL
LIN {X 0,Y 254.382,Z 500.572,A -85,B 0,C 180,E1 -20292.325,E2 -20292.325} C_VEL
LIN {X 0,Y 258.254,Z 485.721,A -85,B 0,C 180,E1 -20293.801,E2 -20293.801} C_VEL
LIN {X 0,Y 261.812,Z 469.529,A -85,B 0,C 180,E1 -20295.065,E2 -20295.065} C_VEL
LIN {X 0,Y 264.836,Z 452.95,A -85,B 0,C 180,E1 -20296.014,E2 -20296.014} C_VEL
LIN {X 0,Y 266.975,Z 436.437,A -85,B 0,C 180,E1 -20296.696,E2 -20296.696} C_VEL
LIN {X 0,Y 268.813,Z 411.5,A -85,B 0,C 180,E1 -20297.395,E2 -20297.395} C_VEL
LIN {X 0,Y 274.972,Z 316.26,A -85,B 0,C 180,E1 -20299.808,E2 -20299.808} C_VEL
LIN {X 0,Y 267.632,Z 300.695,A -85,B 0,C 180,E1 -20302.025,E2 -20302.025} C_VEL
LIN {X 0,Y 257.966,Z 282.54,A -85,B 0,C 180,E1 -20305.155,E2 -20305.155} C_VEL
LIN {X 0,Y 249.228,Z 267.755,A -85,B 0,C 180,E1 -20308.263,E2 -20308.263} C_VEL
LIN {X 0,Y 242.344,Z 258.375,A -85,B 0,C 180,E1 -20310.884,E2 -20310.884} C_VEL
LIN {X 0,Y 239.707,Z 254.891,A -85,B 0,C 180,E1 -20311.948,E2 -20311.948} C_VEL
LIN {X 0,Y 236.378,Z 250.489,A -85,B 0,C 180,E1 -20313.366,E2 -20313.366} C_VEL
LIN {X 0,Y 233.535,Z 246.524,A -85,B 0,C 180,E1 -20314.667,E2 -20314.667} C_VEL
LIN {X 0,Y 230.388,Z 242.9,A -85,B 0,C 180,E1 -20316.141,E2 -20316.141} C_VEL
LIN {X 0,Y 229.417,Z 241.317,A -85,B 0,C 180,E1 -20316.64,E2 -20316.64} C_VEL
LIN {X 0,Y 226.793,Z 238.864,A -85,B 0,C 180,E1 -20317.906,E2 -20317.906} C_VEL
LIN {X 0,Y 225.141,Z 235.893,A -85,B 0,C 180,E1 -20318.843,E2 -20318.843} C_VEL
LIN {X 0,Y 222.613,Z 234.056,A -85,B 0,C 180,E1 -20320.162,E2 -20320.162} C_VEL
LIN {X 0,Y 221.264,Z 231.773,A -85,B 0,C 180,E1 -20321.001,E2 -20321.001} C_VEL
LIN {X 0,Y 220.913,Z 230.242,A -85,B 0,C 180,E1 -20321.331,E2 -20321.331} C_VEL
LIN {X 0,Y 220.97,Z 230.246,A -85,B 0,C 180,E1 -20325.26,E2 -20325.26} C_VEL
LIN {X 0,Y 221.21,Z 230.229,A -85,B 0,C 180,E1 -20330.861,E2 -20330.861} C_VEL
LIN {X 0,Y 221.278,Z 230.227,A -85,B 0,C 180,E1 -20332.702,E2 -20332.702} C_VEL
LIN {X 0,Y 221.485,Z 230.161,A -85,B 0,C 180,E1 -20338.183,E2 -20338.183} C_VEL
LIN {X 0,Y 221.485,Z 230.202,A -85,B 0,C 180,E1 -20341.819,E2 -20341.819} C_VEL
LIN {X 0,Y 221.233,Z 230.233,A -85,B 0,C 180,E1 -20347.301,E2 -20347.301} C_VEL
LIN {X 0,Y 221.039,Z 230.228,A -85,B 0,C 180,E1 -20350.999,E2 -20350.999} C_VEL
LIN {X 0,Y 220.993,Z 230.253,A -85,B 0,C 180,E1 -20356.633,E2 -20356.633} C_VEL
LIN {X 0,Y 220.87,Z 230.258,A -85,B 0,C 180,E1 -20360.489,E2 -20360.489} C_VEL
LIN {X 0,Y 220.846,Z 230.263,A -85,B 0,C 180,E1 -20364.439,E2 -20364.439} C_VEL
LIN {X 0,Y 220.817,Z 230.283,A -85,B 0,C 180,E1 -20368.517,E2 -20368.517} C_VEL
LIN {X 0,Y 220.799,Z 230.262,A -85,B 0,C 180,E1 -20372.76,E2 -20372.76} C_VEL
LIN {X 0,Y 220.793,Z 230.281,A -85,B 0,C 180,E1 -20377.282,E2 -20377.282} C_VEL
LIN {X 0,Y 220.747,Z 230.3,A -85,B 0,C 180,E1 -20381.959,E2 -20381.959} C_VEL
LIN {X 0,Y 220.766,Z 230.419,A -85,B 0,C 180,E1 -20386.175,E2 -20386.175} C_VEL
LIN {X 0,Y 221.487,Z 232.72,A -85,B 0,C 180,E1 -20386.714,E2 -20386.714} C_VEL
LIN {X 0,Y 223.453,Z 235.008,A -85,B 0,C 180,E1 -20387.835,E2 -20387.835} C_VEL
LIN {X 0,Y 225.194,Z 236.194,A -85,B 0,C 180,E1 -20388.722,E2 -20388.722} C_VEL
LIN {X 0,Y 226.986,Z 239.236,A -85,B 0,C 180,E1 -20389.718,E2 -20389.718} C_VEL
LIN {X 0,Y 229.714,Z 241.86,A -85,B 0,C 180,E1 -20391.046,E2 -20391.046} C_VEL
LIN {X 0,Y 232.058,Z 245.215,A -85,B 0,C 180,E1 -20392.205,E2 -20392.205} C_VEL
LIN {X 0,Y 233.883,Z 247.146,A -85,B 0,C 180,E1 -20393.028,E2 -20393.028} C_VEL
LIN {X 0,Y 236.697,Z 250.792,A -85,B 0,C 180,E1 -20394.278,E2 -20394.278} C_VEL
LIN {X 0,Y 241.899,Z 257.755,A -85,B 0,C 180,E1 -20396.461,E2 -20396.461} C_VEL
LIN {X 0,Y 248.059,Z 266.166,A -85,B 0,C 180,E1 -20398.832,E2 -20398.832} C_VEL
LIN {X 0,Y 255.5,Z 276.998,A -85,B 0,C 180,E1 -20401.459,E2 -20401.459} C_VEL
LIN {X 0,Y 264.216,Z 290.782,A -85,B 0,C 180,E1 -20404.277,E2 -20404.277} C_VEL
LIN {X 0,Y 272.74,Z 305.506,A -85,B 0,C 180,E1 -20406.816,E2 -20406.816} C_VEL
LIN {X 0,Y 275.036,Z 309.725,A -85,B 0,C 180,E1 -20407.467,E2 -20407.467} C_VEL
LIN {X 0,Y 267.728,Z 421.758,A -85,B 0,C 180,E1 -20410.351,E2 -20410.351} C_VEL
LIN {X 0,Y 265.564,Z 439.816,A -85,B 0,C 180,E1 -20411.088,E2 -20411.088} C_VEL
LIN {X 0,Y 263.01,Z 455.45,A -85,B 0,C 180,E1 -20412.008,E2 -20412.008} C_VEL
LIN {X 0,Y 260.052,Z 470.05,A -85,B 0,C 180,E1 -20413.115,E2 -20413.115} C_VEL
LIN {X 0,Y 256.68,Z 484.403,A -85,B 0,C 180,E1 -20414.482,E2 -20414.482} C_VEL
LIN {X 0,Y 252.741,Z 498.448,A -85,B 0,C 180,E1 -20416.128,E2 -20416.128} C_VEL
LIN {X 0,Y 248.224,Z 512.599,A -85,B 0,C 180,E1 -20418.159,E2 -20418.159} C_VEL
LIN {X 0,Y 243.713,Z 525.558,A -85,B 0,C 180,E1 -20420.447,E2 -20420.447} C_VEL
LIN {X 0,Y 239.511,Z 536.824,A -85,B 0,C 180,E1 -20422.84,E2 -20422.84} C_VEL
LIN {X 0,Y 235.132,Z 547.979,A -85,B 0,C 180,E1 -20425.719,E2 -20425.719} C_VEL
LIN {X 0,Y 231.224,Z 557.486,A -85,B 0,C 180,E1 -20428.698,E2 -20428.698} C_VEL
LIN {X 0,Y 227.407,Z 566.726,A -85,B 0,C 180,E1 -20432.218,E2 -20432.218} C_VEL
LIN {X 0,Y 224.696,Z 573.575,A -85,B 0,C 180,E1 -20435.388,E2 -20435.388} C_VEL
LIN {X 0,Y 221.905,Z 581.099,A -85,B 0,C 180,E1 -20439.786,E2 -20439.786} C_VEL
LIN {X 0,Y 220.17,Z 586.373,A -85,B 0,C 180,E1 -20443.855,E2 -20443.855} C_VEL
LIN {X 0,Y 219.225,Z 589.36,A -85,B 0,C 180,E1 -20446.774,E2 -20446.774} C_VEL
LIN {X 0,Y 218.383,Z 592.456,A -85,B 0,C 180,E1 -20451.045,E2 -20451.045} C_VEL
LIN {X 0,Y 218.056,Z 594.29,A -85,B 0,C 180,E1 -20455.516,E2 -20455.516} C_VEL
LIN {X 0,Y 218.191,Z 594.761,A -85,B 0,C 180,E1 -20459.577,E2 -20459.577} C_VEL
LIN {X 0,Y 218.498,Z 594.198,A -85,B 0,C 180,E1 -20463.248,E2 -20463.248} C_VEL
LIN {X 0,Y 219.404,Z 592.366,A -85,B 0,C 180,E1 -20467.493,E2 -20467.493} C_VEL
LIN {X 0,Y 221.109,Z 589.127,A -85,B 0,C 180,E1 -20471.877,E2 -20471.877} C_VEL
LIN {X 0,Y 223.656,Z 584.355,A -85,B 0,C 180,E1 -20476.285,E2 -20476.285} C_VEL
LIN {X 0,Y 226.439,Z 579.201,A -85,B 0,C 180,E1 -20479.858,E2 -20479.858} C_VEL
LIN {X 0,Y 230.627,Z 571.854,A -85,B 0,C 180,E1 -20483.823,E2 -20483.823} C_VEL
LIN {X 0,Y 234.746,Z 564.598,A -85,B 0,C 180,E1 -20486.964,E2 -20486.964} C_VEL
LIN {X 0,Y 239.633,Z 555.743,A -85,B 0,C 180,E1 -20490.093,E2 -20490.093} C_VEL
LIN {X 0,Y 244.775,Z 545.975,A -85,B 0,C 180,E1 -20492.887,E2 -20492.887} C_VEL
LIN {X 0,Y 250.688,Z 534.023,A -85,B 0,C 180,E1 -20495.685,E2 -20495.685} C_VEL
LIN {X 0,Y 256.317,Z 521.736,A -85,B 0,C 180,E1 -20498.02,E2 -20498.02} C_VEL
LIN {X 0,Y 261.728,Z 508.783,A -85,B 0,C 180,E1 -20500.028,E2 -20500.028} C_VEL
LIN {X 0,Y 267.131,Z 493.971,A -85,B 0,C 180,E1 -20501.887,E2 -20501.887} C_VEL
LIN {X 0,Y 271.545,Z 480.121,A -85,B 0,C 180,E1 -20503.264,E2 -20503.264} C_VEL
LIN {X 0,Y 275.771,Z 464.319,A -85,B 0,C 180,E1 -20504.541,E2 -20504.541} C_VEL
LIN {X 0,Y 279.197,Z 448.772,A -85,B 0,C 180,E1 -20505.503,E2 -20505.503} C_VEL
LIN {X 0,Y 281.83,Z 433.144,A -85,B 0,C 180,E1 -20506.237,E2 -20506.237} C_VEL
LIN {X 0,Y 283.829,Z 415.744,A -85,B 0,C 180,E1 -20506.785,E2 -20506.785} C_VEL
LIN {X 0,Y 291.561,Z 318.685,A -85,B 0,C 180,E1 -20509.195,E2 -20509.195} C_VEL
LIN {X 0,Y 286.789,Z 309.479,A -85,B 0,C 180,E1 -20511.377,E2 -20511.377} C_VEL
LIN {X 0,Y 282.326,Z 301.803,A -85,B 0,C 180,E1 -20513.642,E2 -20513.642} C_VEL
LIN {X 0,Y 280.45,Z 298.758,A -85,B 0,C 180,E1 -20514.675,E2 -20514.675} C_VEL
LIN {X 0,Y 278.564,Z 296.63,A -85,B 0,C 180,E1 -20515.734,E2 -20515.734} C_VEL
LIN {X 0,Y 275.201,Z 295.122,A -85,B 0,C 180,E1 -20517.637,E2 -20517.637} C_VEL
LIN {X 0,Y 271.587,Z 293.751,A -85,B 0,C 180,E1 -20520.026,E2 -20520.026} C_VEL
LIN {X 0,Y 270.622,Z 292.721,A -85,B 0,C 180,E1 -20520.816,E2 -20520.816} C_VEL
LIN {X 0,Y 268.938,Z 289.781,A -85,B 0,C 180,E1 -20522.506,E2 -20522.506} C_VEL
LIN {X 0,Y 266.731,Z 286.647,A -85,B 0,C 180,E1 -20525.132,E2 -20525.132} C_VEL
LIN {X 0,Y 266.117,Z 285.609,A -85,B 0,C 180,E1 -20526.063,E2 -20526.063} C_VEL
LIN {X 0,Y 263.86,Z 283.52,A -85,B 0,C 180,E1 -20531.485,E2 -20531.485} C_VEL
LIN {X 0,Y 263.754,Z 283.34,A -85,B 0,C 180,E1 -20534.256,E2 -20534.256} C_VEL
LIN {X 0,Y 266.078,Z 285.927,A -85,B 0,C 180,E1 -20540.571,E2 -20540.571} C_VEL
LIN {X 0,Y 267.944,Z 289.293,A -85,B 0,C 180,E1 -20543.168,E2 -20543.168} C_VEL
LIN {X 0,Y 269.192,Z 290.713,A -85,B 0,C 180,E1 -20544.452,E2 -20544.452} C_VEL
LIN {X 0,Y 272.245,Z 295.481,A -85,B 0,C 180,E1 -20547.21,E2 -20547.21} C_VEL
LIN {X 0,Y 275.097,Z 300.431,A -85,B 0,C 180,E1 -20549.363,E2 -20549.363} C_VEL
LIN {X 0,Y 278.137,Z 306.173,A -85,B 0,C 180,E1 -20551.377,E2 -20551.377} C_VEL
LIN {X 0,Y 282.377,Z 314.83,A -85,B 0,C 180,E1 -20553.834,E2 -20553.834} C_VEL
LIN {X 0,Y 286.81,Z 325.016,A -85,B 0,C 180,E1 -20556.13,E2 -20556.13} C_VEL
LIN {X 0,Y 287.506,Z 326.874,A -85,B 0,C 180,E1 -20556.48,E2 -20556.48} C_VEL
LIN {X 0,Y 278.644,Z 431.958,A -85,B 0,C 180,E1 -20559.103,E2 -20559.103} C_VEL
LIN {X 0,Y 275.914,Z 449.721,A -85,B 0,C 180,E1 -20559.738,E2 -20559.738} C_VEL
LIN {X 0,Y 272.397,Z 466.203,A -85,B 0,C 180,E1 -20560.577,E2 -20560.577} C_VEL
LIN {X 0,Y 268.123,Z 482.175,A -85,B 0,C 180,E1 -20561.663,E2 -20561.663} C_VEL
LIN {X 0,Y 263.22,Z 497.628,A -85,B 0,C 180,E1 -20563.034,E2 -20563.034} C_VEL
LIN {X 0,Y 257.947,Z 511.904,A -85,B 0,C 180,E1 -20564.615,E2 -20564.615} C_VEL
LIN {X 0,Y 252.581,Z 524.829,A -85,B 0,C 180,E1 -20566.385,E2 -20566.385} C_VEL
LIN {X 0,Y 246.746,Z 537.526,A -85,B 0,C 180,E1 -20568.527,E2 -20568.527} C_VEL
LIN {X 0,Y 240.609,Z 549.859,A -85,B 0,C 180,E1 -20571.094,E2 -20571.094} C_VEL
LIN {X 0,Y 234.662,Z 561.016,A -85,B 0,C 180,E1 -20573.961,E2 -20573.961} C_VEL
LIN {X 0,Y 229.326,Z 570.727,A -85,B 0,C 180,E1 -20577.042,E2 -20577.042} C_VEL
LIN {X 0,Y 224.385,Z 579.366,A -85,B 0,C 180,E1 -20580.438,E2 -20580.438} C_VEL
LIN {X 0,Y 219.862,Z 587.456,A -85,B 0,C 180,E1 -20584.431,E2 -20584.431} C_VEL
LIN {X 0,Y 216.712,Z 593.374,A -85,B 0,C 180,E1 -20588.099,E2 -20588.099} C_VEL
LIN {X 0,Y 213.901,Z 599.185,A -85,B 0,C 180,E1 -20592.796,E2 -20592.796} C_VEL
LIN {X 0,Y 212.384,Z 602.603,A -85,B 0,C 180,E1 -20596.602,E2 -20596.602} C_VEL
LIN {X 0,Y 211.608,Z 605.093,A -85,B 0,C 180,E1 -20600.437,E2 -20600.437} C_VEL
LIN {X 0,Y 211.369,Z 606.538,A -85,B 0,C 180,E1 -20604.271,E2 -20604.271} C_VEL
LIN {X 0,Y 211.448,Z 607.084,A -85,B 0,C 180,E1 -20608.091,E2 -20608.091} C_VEL
LIN {X 0,Y 211.561,Z 606.957,A -85,B 0,C 180,E1 -20609.995,E2 -20609.995} C_VEL
LIN {X 0,Y 211.441,Z 605.732,A -85,B 0,C 180,E1 -20614.333,E2 -20614.333} C_VEL
LIN {X 0,Y 211.429,Z 603.968,A -85,B 0,C 180,E1 -20617.636,E2 -20617.636} C_VEL
LIN {X 0,Y 211.874,Z 600.886,A -85,B 0,C 180,E1 -20621.475,E2 -20621.475} C_VEL
LIN {X 0,Y 212.941,Z 596.784,A -85,B 0,C 180,E1 -20625.304,E2 -20625.304} C_VEL
LIN {X 0,Y 214.597,Z 591.418,A -85,B 0,C 180,E1 -20629.111,E2 -20629.111} C_VEL
LIN {X 0,Y 216.997,Z 584.845,A -85,B 0,C 180,E1 -20632.865,E2 -20632.865} C_VEL
LIN {X 0,Y 220.353,Z 576.394,A -85,B 0,C 180,E1 -20636.744,E2 -20636.744} C_VEL
LIN {X 0,Y 224.147,Z 567.312,A -85,B 0,C 180,E1 -20640.104,E2 -20640.104} C_VEL
LIN {X 0,Y 228.298,Z 557.371,A -85,B 0,C 180,E1 -20643.115,E2 -20643.115} C_VEL
LIN {X 0,Y 232.956,Z 545.736,A -85,B 0,C 180,E1 -20646.029,E2 -20646.029} C_VEL
LIN {X 0,Y 237.855,Z 533.045,A -85,B 0,C 180,E1 -20648.616,E2 -20648.616} C_VEL
LIN {X 0,Y 242.855,Z 519.22,A -85,B 0,C 180,E1 -20650.893,E2 -20650.893} C_VEL
LIN {X 0,Y 247.638,Z 504.002,A -85,B 0,C 180,E1 -20652.924,E2 -20652.924} C_VEL
LIN {X 0,Y 251.432,Z 490.692,A -85,B 0,C 180,E1 -20654.323,E2 -20654.323} C_VEL
LIN {X 0,Y 255.28,Z 474.593,A -85,B 0,C 180,E1 -20655.701,E2 -20655.701} C_VEL
LIN {X 0,Y 258.448,Z 458.697,A -85,B 0,C 180,E1 -20656.733,E2 -20656.733} C_VEL
LIN {X 0,Y 260.988,Z 442.46,A -85,B 0,C 180,E1 -20657.505,E2 -20657.505} C_VEL
LIN {X 0,Y 262.63,Z 425.765,A -85,B 0,C 180,E1 -20658.059,E2 -20658.059} C_VEL
LIN {X 0,Y 269.764,Z 318.576,A -85,B 0,C 180,E1 -20660.82,E2 -20660.82} C_VEL
LIN {X 0,Y 261.839,Z 301.966,A -85,B 0,C 180,E1 -20663.331,E2 -20663.331} C_VEL
LIN {X 0,Y 253.548,Z 286.322,A -85,B 0,C 180,E1 -20666.154,E2 -20666.154} C_VEL
LIN {X 0,Y 245.501,Z 272.666,A -85,B 0,C 180,E1 -20669.134,E2 -20669.134} C_VEL
LIN {X 0,Y 237.601,Z 261.636,A -85,B 0,C 180,E1 -20672.294,E2 -20672.294} C_VEL
LIN {X 0,Y 233.233,Z 255.986,A -85,B 0,C 180,E1 -20674.209,E2 -20674.209} C_VEL
LIN {X 0,Y 230.078,Z 251.724,A -85,B 0,C 180,E1 -20675.707,E2 -20675.707} C_VEL
LIN {X 0,Y 227.381,Z 248.279,A -85,B 0,C 180,E1 -20677.033,E2 -20677.033} C_VEL
LIN {X 0,Y 223.867,Z 244.294,A -85,B 0,C 180,E1 -20678.838,E2 -20678.838} C_VEL
LIN {X 0,Y 222.623,Z 242.258,A -85,B 0,C 180,E1 -20679.561,E2 -20679.561} C_VEL
LIN {X 0,Y 219.94,Z 239.773,A -85,B 0,C 180,E1 -20681.064,E2 -20681.064} C_VEL
LIN {X 0,Y 218.407,Z 236.881,A -85,B 0,C 180,E1 -20682.08,E2 -20682.08} C_VEL
LIN {X 0,Y 215.704,Z 235.016,A -85,B 0,C 180,E1 -20683.68,E2 -20683.68} C_VEL
LIN {X 0,Y 214.313,Z 232.727,A -85,B 0,C 180,E1 -20684.67,E2 -20684.67} C_VEL
LIN {X 0,Y 213.927,Z 231.125,A -85,B 0,C 180,E1 -20685.129,E2 -20685.129} C_VEL
LIN {X 0,Y 214.142,Z 231.101,A -85,B 0,C 180,E1 -20690.556,E2 -20690.556} C_VEL
LIN {X 0,Y 214.213,Z 231.111,A -85,B 0,C 180,E1 -20692.46,E2 -20692.46} C_VEL
LIN {X 0,Y 214.418,Z 231.039,A -85,B 0,C 180,E1 -20698.123,E2 -20698.123} C_VEL
LIN {X 0,Y 214.524,Z 231.066,A -85,B 0,C 180,E1 -20700.001,E2 -20700.001} C_VEL
LIN {X 0,Y 214.418,Z 231.081,A -85,B 0,C 180,E1 -20701.879,E2 -20701.879} C_VEL
LIN {X 0,Y 214.173,Z 231.115,A -85,B 0,C 180,E1 -20707.543,E2 -20707.543} C_VEL
LIN {X 0,Y 213.971,Z 231.106,A -85,B 0,C 180,E1 -20711.367,E2 -20711.367} C_VEL
LIN {X 0,Y 213.906,Z 231.15,A -85,B 0,C 180,E1 -20715.24,E2 -20715.24} C_VEL
LIN {X 0,Y 213.817,Z 231.126,A -85,B 0,C 180,E1 -20719.191,E2 -20719.191} C_VEL
LIN {X 0,Y 213.827,Z 231.156,A -85,B 0,C 180,E1 -20723.23,E2 -20723.23} C_VEL
LIN {X 0,Y 213.81,Z 231.137,A -85,B 0,C 180,E1 -20727.454,E2 -20727.454} C_VEL
LIN {X 0,Y 213.75,Z 231.144,A -85,B 0,C 180,E1 -20731.742,E2 -20731.742} C_VEL
LIN {X 0,Y 213.727,Z 231.176,A -85,B 0,C 180,E1 -20736.293,E2 -20736.293} C_VEL
LIN {X 0,Y 213.69,Z 231.164,A -85,B 0,C 180,E1 -20741.132,E2 -20741.132} C_VEL
LIN {X 0,Y 213.732,Z 231.312,A -85,B 0,C 180,E1 -20742.385,E2 -20742.385} C_VEL
LIN {X 0,Y 214.408,Z 233.452,A -85,B 0,C 180,E1 -20742.974,E2 -20742.974} C_VEL
LIN {X 0,Y 216.065,Z 235.626,A -85,B 0,C 180,E1 -20744.098,E2 -20744.098} C_VEL
LIN {X 0,Y 218.402,Z 237.219,A -85,B 0,C 180,E1 -20745.479,E2 -20745.479} C_VEL
LIN {X 0,Y 220.105,Z 240.236,A -85,B 0,C 180,E1 -20746.588,E2 -20746.588} C_VEL
LIN {X 0,Y 222.919,Z 242.878,A -85,B 0,C 180,E1 -20748.148,E2 -20748.148} C_VEL
LIN {X 0,Y 225.361,Z 246.31,A -85,B 0,C 180,E1 -20749.489,E2 -20749.489} C_VEL
LIN {X 0,Y 227.224,Z 248.096,A -85,B 0,C 180,E1 -20750.413,E2 -20750.413} C_VEL
LIN {X 0,Y 229.798,Z 251.61,A -85,B 0,C 180,E1 -20751.704,E2 -20751.704} C_VEL
LIN {X 0,Y 231.414,Z 253.519,A -85,B 0,C 180,E1 -20752.466,E2 -20752.466} C_VEL
LIN {X 0,Y 235.105,Z 258.412,A -85,B 0,C 180,E1 -20754.145,E2 -20754.145} C_VEL
LIN {X 0,Y 241.297,Z 266.703,A -85,B 0,C 180,E1 -20756.746,E2 -20756.746} C_VEL
LIN {X 0,Y 249.739,Z 278.894,A -85,B 0,C 180,E1 -20759.954,E2 -20759.954} C_VEL
LIN {X 0,Y 258.47,Z 292.6,A -85,B 0,C 180,E1 -20762.947,E2 -20762.947} C_VEL
LIN {X 0,Y 267.3,Z 307.736,A -85,B 0,C 180,E1 -20765.705,E2 -20765.705} C_VEL
LIN {X 0,Y 269.943,Z 312.904,A -85,B 0,C 180,E1 -20766.505,E2 -20766.505} C_VEL
LIN {X 0,Y 262.468,Z 422.086,A -85,B 0,C 180,E1 -20769.326,E2 -20769.326} C_VEL
LIN {X 0,Y 260.246,Z 440.092,A -85,B 0,C 180,E1 -20770.071,E2 -20770.071} C_VEL
LIN {X 0,Y 257.39,Z 456.983,A -85,B 0,C 180,E1 -20771.085,E2 -20771.085} C_VEL
LIN {X 0,Y 254.151,Z 472.242,A -85,B 0,C 180,E1 -20772.296,E2 -20772.296} C_VEL
LIN {X 0,Y 250.139,Z 487.87,A -85,B 0,C 180,E1 -20773.855,E2 -20773.855} C_VEL
LIN {X 0,Y 246.147,Z 501.461,A -85,B 0,C 180,E1 -20775.537,E2 -20775.537} C_VEL
LIN {X 0,Y 241.555,Z 515.214,A -85,B 0,C 180,E1 -20777.614,E2 -20777.614} C_VEL
LIN {X 0,Y 236.633,Z 528.545,A -85,B 0,C 180,E1 -20780.104,E2 -20780.104} C_VEL
LIN {X 0,Y 232.31,Z 539.57,A -85,B 0,C 180,E1 -20782.617,E2 -20782.617} C_VEL
LIN {X 0,Y 227.853,Z 550.381,A -85,B 0,C 180,E1 -20785.582,E2 -20785.582} C_VEL
LIN {X 0,Y 223.915,Z 559.649,A -85,B 0,C 180,E1 -20788.656,E2 -20788.656} C_VEL
LIN {X 0,Y 220.066,Z 568.55,A -85,B 0,C 180,E1 -20792.292,E2 -20792.292} C_VEL
LIN {X 0,Y 217.368,Z 575.103,A -85,B 0,C 180,E1 -20795.571,E2 -20795.571} C_VEL
LIN {X 0,Y 214.947,Z 581.379,A -85,B 0,C 180,E1 -20799.413,E2 -20799.413} C_VEL
LIN {X 0,Y 213.22,Z 586.333,A -85,B 0,C 180,E1 -20803.344,E2 -20803.344} C_VEL
LIN {X 0,Y 211.971,Z 590.188,A -85,B 0,C 180,E1 -20807.366,E2 -20807.366} C_VEL
LIN {X 0,Y 211.232,Z 592.953,A -85,B 0,C 180,E1 -20811.472,E2 -20811.472} C_VEL
LIN {X 0,Y 210.958,Z 594.576,A -85,B 0,C 180,E1 -20815.906,E2 -20815.906} C_VEL
LIN {X 0,Y 211.104,Z 594.955,A -85,B 0,C 180,E1 -20820.049,E2 -20820.049} C_VEL
LIN {X 0,Y 211.586,Z 594.212,A -85,B 0,C 180,E1 -20824.383,E2 -20824.383} C_VEL
LIN {X 0,Y 212.775,Z 592.083,A -85,B 0,C 180,E1 -20828.875,E2 -20828.875} C_VEL
LIN {X 0,Y 214.759,Z 588.523,A -85,B 0,C 180,E1 -20833.415,E2 -20833.415} C_VEL
LIN {X 0,Y 217.669,Z 583.409,A -85,B 0,C 180,E1 -20837.959,E2 -20837.959} C_VEL
LIN {X 0,Y 220.595,Z 578.528,A -85,B 0,C 180,E1 -20841.315,E2 -20841.315} C_VEL
LIN {X 0,Y 225.086,Z 571.12,A -85,B 0,C 180,E1 -20845.275,E2 -20845.275} C_VEL
LIN {X 0,Y 230.042,Z 562.737,A -85,B 0,C 180,E1 -20848.811,E2 -20848.811} C_VEL
LIN {X 0,Y 235.407,Z 553.389,A -85,B 0,C 180,E1 -20851.988,E2 -20851.988} C_VEL
LIN {X 0,Y 240.894,Z 543.445,A -85,B 0,C 180,E1 -20854.749,E2 -20854.749} C_VEL
LIN {X 0,Y 247.164,Z 531.043,A -85,B 0,C 180,E1 -20857.542,E2 -20857.542} C_VEL
LIN {X 0,Y 253.369,Z 517.644,A -85,B 0,C 180,E1 -20859.936,E2 -20859.936} C_VEL
LIN {X 0,Y 258.866,Z 504.37,A -85,B 0,C 180,E1 -20861.851,E2 -20861.851} C_VEL
LIN {X 0,Y 263.91,Z 490.59,A -85,B 0,C 180,E1 -20863.479,E2 -20863.479} C_VEL
LIN {X 0,Y 268.459,Z 476.446,A -85,B 0,C 180,E1 -20864.823,E2 -20864.823} C_VEL
LIN {X 0,Y 272.545,Z 461.053,A -85,B 0,C 180,E1 -20865.988,E2 -20865.988} C_VEL
LIN {X 0,Y 275.415,Z 447.658,A -85,B 0,C 180,E1 -20866.782,E2 -20866.782} C_VEL
LIN {X 0,Y 278.143,Z 431.467,A -85,B 0,C 180,E1 -20867.511,E2 -20867.511} C_VEL
LIN {X 0,Y 280.075,Z 414.671,A -85,B 0,C 180,E1 -20868.022,E2 -20868.022} C_VEL
LIN {X 0,Y 287.737,Z 322.177,A -85,B 0,C 180,E1 -20870.323,E2 -20870.323} C_VEL
LIN {X 0,Y 283.784,Z 314.473,A -85,B 0,C 180,E1 -20872.241,E2 -20872.241} C_VEL
LIN {X 0,Y 279.636,Z 307.13,A -85,B 0,C 180,E1 -20874.484,E2 -20874.484} C_VEL
LIN {X 0,Y 275.616,Z 300.37,A -85,B 0,C 180,E1 -20876.988,E2 -20876.988} C_VEL
LIN {X 0,Y 273.819,Z 297.547,A -85,B 0,C 180,E1 -20878.24,E2 -20878.24} C_VEL
LIN {X 0,Y 271.468,Z 293.91,A -85,B 0,C 180,E1 -20880.092,E2 -20880.092} C_VEL
LIN {X 0,Y 270.622,Z 292.721,A -85,B 0,C 180,E1 -20880.816,E2 -20880.816} C_VEL
LIN {X 0,Y 269.285,Z 291.502,A -85,B 0,C 180,E1 -20882.008,E2 -20882.008} C_VEL
LIN {X 0,Y 267.909,Z 291.305,A -85,B 0,C 180,E1 -20883.239,E2 -20883.239} C_VEL
LIN {X 0,Y 264.795,Z 292.273,A -85,B 0,C 180,E1 -20886.619,E2 -20886.619} C_VEL
LIN {X 0,Y 264.255,Z 292.1,A -85,B 0,C 180,E1 -20887.479,E2 -20887.479} C_VEL
LIN {X 0,Y 262.898,Z 290.552,A -85,B 0,C 180,E1 -20891.527,E2 -20891.527} C_VEL
LIN {X 0,Y 262.802,Z 290.399,A -85,B 0,C 180,E1 -20894.309,E2 -20894.309} C_VEL
LIN {X 0,Y 264.895,Z 292.818,A -85,B 0,C 180,E1 -20900.256,E2 -20900.256} C_VEL
LIN {X 0,Y 266.791,Z 296.242,A -85,B 0,C 180,E1 -20902.989,E2 -20902.989} C_VEL
LIN {X 0,Y 267.834,Z 297.517,A -85,B 0,C 180,E1 -20904.101,E2 -20904.101} C_VEL
LIN {X 0,Y 270.747,Z 302.234,A -85,B 0,C 180,E1 -20906.847,E2 -20906.847} C_VEL
LIN {X 0,Y 273.267,Z 306.914,A -85,B 0,C 180,E1 -20908.856,E2 -20908.856} C_VEL
LIN {X 0,Y 276.117,Z 312.416,A -85,B 0,C 180,E1 -20910.82,E2 -20910.82} C_VEL
LIN {X 0,Y 279.821,Z 320.417,A -85,B 0,C 180,E1 -20913.101,E2 -20913.101} C_VEL
LIN {X 0,Y 283.776,Z 329.84,A -85,B 0,C 180,E1 -20915.283,E2 -20915.283} C_VEL
LIN {X 0,Y 274.939,Z 431.464,A -85,B 0,C 180,E1 -20917.841,E2 -20917.841} C_VEL
LIN {X 0,Y 272.201,Z 448.915,A -85,B 0,C 180,E1 -20918.462,E2 -20918.462} C_VEL
LIN {X 0,Y 268.819,Z 464.503,A -85,B 0,C 180,E1 -20919.236,E2 -20919.236} C_VEL
LIN {X 0,Y 264.708,Z 479.842,A -85,B 0,C 180,E1 -20920.24,E2 -20920.24} C_VEL
LIN {X 0,Y 260.15,Z 494.179,A -85,B 0,C 180,E1 -20921.435,E2 -20921.435} C_VEL
LIN {X 0,Y 254.69,Z 508.907,A -85,B 0,C 180,E1 -20923.006,E2 -20923.006} C_VEL
LIN {X 0,Y 248.894,Z 522.533,A -85,B 0,C 180,E1 -20924.806,E2 -20924.806} C_VEL
LIN {X 0,Y 243.432,Z 534.261,A -85,B 0,C 180,E1 -20926.708,E2 -20926.708} C_VEL
LIN {X 0,Y 236.881,Z 547.073,A -85,B 0,C 180,E1 -20929.25,E2 -20929.25} C_VEL
LIN {X 0,Y 230.891,Z 557.944,A -85,B 0,C 180,E1 -20931.944,E2 -20931.944} C_VEL
LIN {X 0,Y 224.809,Z 568.539,A -85,B 0,C 180,E1 -20935.209,E2 -20935.209} C_VEL
LIN {X 0,Y 219.409,Z 577.503,A -85,B 0,C 180,E1 -20938.63,E2 -20938.63} C_VEL
LIN {X 0,Y 215.364,Z 584.222,A -85,B 0,C 180,E1 -20941.773,E2 -20941.773} C_VEL
LIN {X 0,Y 211.615,Z 590.602,A -85,B 0,C 180,E1 -20945.468,E2 -20945.468} C_VEL
LIN {X 0,Y 208.678,Z 595.911,A -85,B 0,C 180,E1 -20949.287,E2 -20949.287} C_VEL
LIN {X 0,Y 206.122,Z 600.962,A -85,B 0,C 180,E1 -20954.167,E2 -20954.167} C_VEL
LIN {X 0,Y 204.867,Z 603.841,A -85,B 0,C 180,E1 -20958.117,E2 -20958.117} C_VEL
LIN {X 0,Y 204.355,Z 605.8,A -85,B 0,C 180,E1 -20962.089,E2 -20962.089} C_VEL
LIN {X 0,Y 204.314,Z 606.726,A -85,B 0,C 180,E1 -20966.051,E2 -20966.051} C_VEL
LIN {X 0,Y 204.478,Z 606.739,A -85,B 0,C 180,E1 -20969.995,E2 -20969.995} C_VEL
LIN {X 0,Y 204.342,Z 605.602,A -85,B 0,C 180,E1 -20974.139,E2 -20974.139} C_VEL
LIN {X 0,Y 204.361,Z 603.673,A -85,B 0,C 180,E1 -20977.902,E2 -20977.902} C_VEL
LIN {X 0,Y 204.844,Z 600.534,A -85,B 0,C 180,E1 -20981.874,E2 -20981.874} C_VEL
LIN {X 0,Y 206.017,Z 596.379,A -85,B 0,C 180,E1 -20985.832,E2 -20985.832} C_VEL
LIN {X 0,Y 207.789,Z 590.97,A -85,B 0,C 180,E1 -20989.763,E2 -20989.763} C_VEL
LIN {X 0,Y 210.363,Z 584.324,A -85,B 0,C 180,E1 -20993.629,E2 -20993.629} C_VEL
LIN {X 0,Y 213.7,Z 576.302,A -85,B 0,C 180,E1 -20997.408,E2 -20997.408} C_VEL
LIN {X 0,Y 217.912,Z 566.663,A -85,B 0,C 180,E1 -21001.059,E2 -21001.059} C_VEL
LIN {X 0,Y 222.239,Z 556.626,A -85,B 0,C 180,E1 -21004.14,E2 -21004.14} C_VEL
LIN {X 0,Y 227.155,Z 544.889,A -85,B 0,C 180,E1 -21007.101,E2 -21007.101} C_VEL
LIN {X 0,Y 232.233,Z 532.065,A -85,B 0,C 180,E1 -21009.732,E2 -21009.732} C_VEL
LIN {X 0,Y 236.903,Z 519.649,A -85,B 0,C 180,E1 -21011.807,E2 -21011.807} C_VEL
LIN {X 0,Y 241.489,Z 505.681,A -85,B 0,C 180,E1 -21013.717,E2 -21013.717} C_VEL
LIN {X 0,Y 245.357,Z 492.79,A -85,B 0,C 180,E1 -21015.141,E2 -21015.141} C_VEL
LIN {X 0,Y 249.323,Z 477.322,A -85,B 0,C 180,E1 -21016.531,E2 -21016.531} C_VEL
LIN {X 0,Y 252.625,Z 461.523,A -85,B 0,C 180,E1 -21017.635,E2 -21017.635} C_VEL
LIN {X 0,Y 255.433,Z 445.024,A -85,B 0,C 180,E1 -21018.451,E2 -21018.451} C_VEL
LIN {X 0,Y 257.259,Z 428.579,A -85,B 0,C 180,E1 -21019.042,E2 -21019.042} C_VEL
LIN {X 0,Y 264.731,Z 321.239,A -85,B 0,C 180,E1 -21021.837,E2 -21021.837} C_VEL
LIN {X 0,Y 257.677,Z 306.339,A -85,B 0,C 180,E1 -21024.159,E2 -21024.159} C_VEL
LIN {X 0,Y 249.534,Z 290.77,A -85,B 0,C 180,E1 -21027.05,E2 -21027.05} C_VEL
LIN {X 0,Y 242.161,Z 278.049,A -85,B 0,C 180,E1 -21029.899,E2 -21029.899} C_VEL
LIN {X 0,Y 234.442,Z 267.153,A -85,B 0,C 180,E1 -21033.098,E2 -21033.098} C_VEL
LIN {X 0,Y 230.1,Z 261.436,A -85,B 0,C 180,E1 -21035.092,E2 -21035.092} C_VEL
LIN {X 0,Y 227.564,Z 257.905,A -85,B 0,C 180,E1 -21036.33,E2 -21036.33} C_VEL
LIN {X 0,Y 224.08,Z 253.519,A -85,B 0,C 180,E1 -21038.104,E2 -21038.104} C_VEL
LIN {X 0,Y 221.304,Z 250.184,A -85,B 0,C 180,E1 -21039.615,E2 -21039.615} C_VEL
LIN {X 0,Y 220.344,Z 248.662,A -85,B 0,C 180,E1 -21040.192,E2 -21040.192} C_VEL
LIN {X 0,Y 217.6,Z 245.87,A -85,B 0,C 180,E1 -21041.793,E2 -21041.793} C_VEL
LIN {X 0,Y 216.116,Z 243.338,A -85,B 0,C 180,E1 -21042.777,E2 -21042.777} C_VEL
LIN {X 0,Y 213.563,Z 241.282,A -85,B 0,C 180,E1 -21044.37,E2 -21044.37} C_VEL
LIN {X 0,Y 211.929,Z 238.469,A -85,B 0,C 180,E1 -21045.599,E2 -21045.599} C_VEL
LIN {X 0,Y 211.66,Z 237.827,A -85,B 0,C 180,E1 -21045.826,E2 -21045.826} C_VEL
LIN {X 0,Y 208.993,Z 236.198,A -85,B 0,C 180,E1 -21047.745,E2 -21047.745} C_VEL
LIN {X 0,Y 207.508,Z 233.925,A -85,B 0,C 180,E1 -21049.021,E2 -21049.021} C_VEL
LIN {X 0,Y 207.045,Z 231.966,A -85,B 0,C 180,E1 -21049.644,E2 -21049.644} C_VEL
LIN {X 0,Y 207.152,Z 231.993,A -85,B 0,C 180,E1 -21052.201,E2 -21052.201} C_VEL
LIN {X 0,Y 207.355,Z 231.917,A -85,B 0,C 180,E1 -21058.059,E2 -21058.059} C_VEL
LIN {X 0,Y 207.489,Z 231.941,A -85,B 0,C 180,E1 -21060.001,E2 -21060.001} C_VEL
LIN {X 0,Y 207.355,Z 231.958,A -85,B 0,C 180,E1 -21061.943,E2 -21061.943} C_VEL
LIN {X 0,Y 207.116,Z 231.997,A -85,B 0,C 180,E1 -21067.802,E2 -21067.802} C_VEL
LIN {X 0,Y 206.896,Z 231.986,A -85,B 0,C 180,E1 -21071.761,E2 -21071.761} C_VEL
LIN {X 0,Y 206.841,Z 232.028,A -85,B 0,C 180,E1 -21075.774,E2 -21075.774} C_VEL
LIN {X 0,Y 206.763,Z 232.007,A -85,B 0,C 180,E1 -21079.872,E2 -21079.872} C_VEL
LIN {X 0,Y 206.743,Z 232.022,A -85,B 0,C 180,E1 -21084.076,E2 -21084.076} C_VEL
LIN {X 0,Y 206.725,Z 232.034,A -85,B 0,C 180,E1 -21088.423,E2 -21088.423} C_VEL
LIN {X 0,Y 206.681,Z 232.019,A -85,B 0,C 180,E1 -21092.962,E2 -21092.962} C_VEL
LIN {X 0,Y 206.695,Z 232.114,A -85,B 0,C 180,E1 -21097.738,E2 -21097.738} C_VEL
LIN {X 0,Y 207.358,Z 234.337,A -85,B 0,C 180,E1 -21098.462,E2 -21098.462} C_VEL
LIN {X 0,Y 209.179,Z 236.665,A -85,B 0,C 180,E1 -21099.955,E2 -21099.955} C_VEL
LIN {X 0,Y 211.607,Z 238.224,A -85,B 0,C 180,E1 -21101.7,E2 -21101.7} C_VEL
LIN {X 0,Y 213.3,Z 241.286,A -85,B 0,C 180,E1 -21103.002,E2 -21103.002} C_VEL
LIN {X 0,Y 216.221,Z 243.795,A -85,B 0,C 180,E1 -21104.844,E2 -21104.844} C_VEL
LIN {X 0,Y 218.476,Z 247.2,A -85,B 0,C 180,E1 -21106.297,E2 -21106.297} C_VEL
LIN {X 0,Y 220.692,Z 249.373,A -85,B 0,C 180,E1 -21107.56,E2 -21107.56} C_VEL
LIN {X 0,Y 223.343,Z 252.906,A -85,B 0,C 180,E1 -21109.046,E2 -21109.046} C_VEL
LIN {X 0,Y 224.809,Z 254.441,A -85,B 0,C 180,E1 -21109.797,E2 -21109.797} C_VEL
LIN {X 0,Y 227.569,Z 258.069,A -85,B 0,C 180,E1 -21111.211,E2 -21111.211} C_VEL
LIN {X 0,Y 232.339,Z 264.396,A -85,B 0,C 180,E1 -21113.481,E2 -21113.481} C_VEL
LIN {X 0,Y 238.114,Z 272.221,A -85,B 0,C 180,E1 -21115.989,E2 -21115.989} C_VEL
LIN {X 0,Y 246.607,Z 284.676,A -85,B 0,C 180,E1 -21119.33,E2 -21119.33} C_VEL
LIN {X 0,Y 255.47,Z 298.891,A -85,B 0,C 180,E1 -21122.459,E2 -21122.459} C_VEL
LIN {X 0,Y 263.755,Z 313.425,A -85,B 0,C 180,E1 -21125.126,E2 -21125.126} C_VEL
LIN {X 0,Y 264.756,Z 315.327,A -85,B 0,C 180,E1 -21125.435,E2 -21125.435} C_VEL
LIN {X 0,Y 257.397,Z 421.335,A -85,B 0,C 180,E1 -21128.228,E2 -21128.228} C_VEL
LIN {X 0,Y 255.407,Z 437.729,A -85,B 0,C 180,E1 -21128.893,E2 -21128.893} C_VEL
LIN {X 0,Y 252.789,Z 453.374,A -85,B 0,C 180,E1 -21129.775,E2 -21129.775} C_VEL
LIN {X 0,Y 249.645,Z 468.531,A -85,B 0,C 180,E1 -21130.902,E2 -21130.902} C_VEL
LIN {X 0,Y 245.882,Z 483.551,A -85,B 0,C 180,E1 -21132.325,E2 -21132.325} C_VEL
LIN {X 0,Y 241.5,Z 498.372,A -85,B 0,C 180,E1 -21134.087,E2 -21134.087} C_VEL
LIN {X 0,Y 236.974,Z 511.861,A -85,B 0,C 180,E1 -21136.061,E2 -21136.061} C_VEL
LIN {X 0,Y 232.478,Z 524.089,A -85,B 0,C 180,E1 -21138.23,E2 -21138.23} C_VEL
LIN {X 0,Y 227.916,Z 535.471,A -85,B 0,C 180,E1 -21140.669,E2 -21140.669} C_VEL
LIN {X 0,Y 223.071,Z 546.948,A -85,B 0,C 180,E1 -21143.674,E2 -21143.674} C_VEL
LIN {X 0,Y 218.446,Z 557.454,A -85,B 0,C 180,E1 -21147.051,E2 -21147.051} C_VEL
LIN {X 0,Y 214.56,Z 566.158,A -85,B 0,C 180,E1 -21150.474,E2 -21150.474} C_VEL
LIN {X 0,Y 210.831,Z 574.734,A -85,B 0,C 180,E1 -21154.689,E2 -21154.689} C_VEL
LIN {X 0,Y 208.157,Z 581.233,A -85,B 0,C 180,E1 -21158.743,E2 -21158.743} C_VEL
LIN {X 0,Y 206.307,Z 586.268,A -85,B 0,C 180,E1 -21162.797,E2 -21162.797} C_VEL
LIN {X 0,Y 205.126,Z 589.782,A -85,B 0,C 180,E1 -21166.392,E2 -21166.392} C_VEL
LIN {X 0,Y 204.124,Z 593.248,A -85,B 0,C 180,E1 -21171.623,E2 -21171.623} C_VEL
LIN {X 0,Y 203.862,Z 594.938,A -85,B 0,C 180,E1 -21176.63,E2 -21176.63} C_VEL
LIN {X 0,Y 204.055,Z 595.116,A -85,B 0,C 180,E1 -21181.11,E2 -21181.11} C_VEL
LIN {X 0,Y 204.751,Z 594.08,A -85,B 0,C 180,E1 -21185.703,E2 -21185.703} C_VEL
LIN {X 0,Y 206.196,Z 591.72,A -85,B 0,C 180,E1 -21190.365,E2 -21190.365} C_VEL
LIN {X 0,Y 208.534,Z 587.917,A -85,B 0,C 180,E1 -21195.056,E2 -21195.056} C_VEL
LIN {X 0,Y 211.904,Z 582.496,A -85,B 0,C 180,E1 -21199.718,E2 -21199.718} C_VEL
LIN {X 0,Y 215.177,Z 577.285,A -85,B 0,C 180,E1 -21203.137,E2 -21203.137} C_VEL
LIN {X 0,Y 220.167,Z 569.603,A -85,B 0,C 180,E1 -21207.134,E2 -21207.134} C_VEL
LIN {X 0,Y 225.604,Z 560.901,A -85,B 0,C 180,E1 -21210.726,E2 -21210.726} C_VEL
LIN {X 0,Y 231.135,Z 551.627,A -85,B 0,C 180,E1 -21213.77,E2 -21213.77} C_VEL
LIN {X 0,Y 237.281,Z 540.729,A -85,B 0,C 180,E1 -21216.667,E2 -21216.667} C_VEL
LIN {X 0,Y 243.305,Z 529.117,A -85,B 0,C 180,E1 -21219.187,E2 -21219.187} C_VEL
LIN {X 0,Y 249.34,Z 516.508,A -85,B 0,C 180,E1 -21221.405,E2 -21221.405} C_VEL
LIN {X 0,Y 255.575,Z 501.802,A -85,B 0,C 180,E1 -21223.477,E2 -21223.477} C_VEL
LIN {X 0,Y 261.024,Z 486.935,A -85,B 0,C 180,E1 -21225.136,E2 -21225.136} C_VEL
LIN {X 0,Y 265.517,Z 472.567,A -85,B 0,C 180,E1 -21226.41,E2 -21226.41} C_VEL
LIN {X 0,Y 269.728,Z 456.015,A -85,B 0,C 180,E1 -21227.591,E2 -21227.591} C_VEL
LIN {X 0,Y 273.145,Z 439.21,A -85,B 0,C 180,E1 -21228.455,E2 -21228.455} C_VEL
LIN {X 0,Y 275.506,Z 423.376,A -85,B 0,C 180,E1 -21229.033,E2 -21229.033} C_VEL
LIN {X 0,Y 284,Z 325.653,A -85,B 0,C 180,E1 -21231.5,E2 -21231.5} C_VEL
LIN {X 0,Y 280.043,Z 317.79,A -85,B 0,C 180,E1 -21233.601,E2 -21233.601} C_VEL
LIN {X 0,Y 275.8,Z 310.337,A -85,B 0,C 180,E1 -21236.129,E2 -21236.129} C_VEL
LIN {X 0,Y 272.387,Z 304.411,A -85,B 0,C 180,E1 -21238.521,E2 -21238.521} C_VEL
LIN {X 0,Y 269.594,Z 300.076,A -85,B 0,C 180,E1 -21240.809,E2 -21240.809} C_VEL
LIN {X 0,Y 267.44,Z 296.432,A -85,B 0,C 180,E1 -21243.012,E2 -21243.012} C_VEL
LIN {X 0,Y 265.255,Z 292.871,A -85,B 0,C 180,E1 -21245.89,E2 -21245.89} C_VEL
LIN {X 0,Y 264.255,Z 292.1,A -85,B 0,C 180,E1 -21247.479,E2 -21247.479} C_VEL
LIN {X 0,Y 263.574,Z 292.188,A -85,B 0,C 180,E1 -21248.753,E2 -21248.753} C_VEL
LIN {X 0,Y 262.543,Z 294.181,A -85,B 0,C 180,E1 -21250.855,E2 -21250.855} C_VEL
LIN {X 0,Y 261.853,Z 296.992,A -85,B 0,C 180,E1 -21253.401,E2 -21253.401} C_VEL
LIN {X 0,Y 261.844,Z 297.43,A -85,B 0,C 180,E1 -21254.268,E2 -21254.268} C_VEL
LIN {X 0,Y 263.759,Z 299.803,A -85,B 0,C 180,E1 -21260.009,E2 -21260.009} C_VEL
LIN {X 0,Y 265.817,Z 303.433,A -85,B 0,C 180,E1 -21263.011,E2 -21263.011} C_VEL
LIN {X 0,Y 266.575,Z 304.516,A -85,B 0,C 180,E1 -21263.85,E2 -21263.85} C_VEL
LIN {X 0,Y 269.113,Z 308.78,A -85,B 0,C 180,E1 -21266.356,E2 -21266.356} C_VEL
LIN {X 0,Y 271.356,Z 313.066,A -85,B 0,C 180,E1 -21268.235,E2 -21268.235} C_VEL
LIN {X 0,Y 274.352,Z 319.184,A -85,B 0,C 180,E1 -21270.416,E2 -21270.416} C_VEL
LIN {X 0,Y 277.594,Z 326.708,A -85,B 0,C 180,E1 -21272.529,E2 -21272.529} C_VEL
LIN {X 0,Y 280.233,Z 333.238,A -85,B 0,C 180,E1 -21274.089,E2 -21274.089} C_VEL
LIN {X 0,Y 271.446,Z 430.739,A -85,B 0,C 180,E1 -21276.538,E2 -21276.538} C_VEL
LIN {X 0,Y 268.782,Z 447.67,A -85,B 0,C 180,E1 -21277.132,E2 -21277.132} C_VEL
LIN {X 0,Y 265.386,Z 463.074,A -85,B 0,C 180,E1 -21277.858,E2 -21277.858} C_VEL
LIN {X 0,Y 261.432,Z 477.684,A -85,B 0,C 180,E1 -21278.773,E2 -21278.773} C_VEL
LIN {X 0,Y 256.717,Z 492.199,A -85,B 0,C 180,E1 -21279.953,E2 -21279.953} C_VEL
LIN {X 0,Y 251.047,Z 507.179,A -85,B 0,C 180,E1 -21281.505,E2 -21281.505} C_VEL
LIN {X 0,Y 245.03,Z 521.065,A -85,B 0,C 180,E1 -21283.294,E2 -21283.294} C_VEL
LIN {X 0,Y 239.322,Z 533.002,A -85,B 0,C 180,E1 -21285.184,E2 -21285.184} C_VEL
LIN {X 0,Y 232.494,Z 545.903,A -85,B 0,C 180,E1 -21287.729,E2 -21287.729} C_VEL
LIN {X 0,Y 226.183,Z 556.873,A -85,B 0,C 180,E1 -21290.429,E2 -21290.429} C_VEL
LIN {X 0,Y 220.533,Z 566.372,A -85,B 0,C 180,E1 -21293.303,E2 -21293.303} C_VEL
LIN {X 0,Y 214.658,Z 575.679,A -85,B 0,C 180,E1 -21296.739,E2 -21296.739} C_VEL
LIN {X 0,Y 209.273,Z 584.019,A -85,B 0,C 180,E1 -21300.663,E2 -21300.663} C_VEL
LIN {X 0,Y 205.087,Z 590.654,A -85,B 0,C 180,E1 -21304.633,E2 -21304.633} C_VEL
LIN {X 0,Y 201.959,Z 595.909,A -85,B 0,C 180,E1 -21308.564,E2 -21308.564} C_VEL
LIN {X 0,Y 199.217,Z 600.916,A -85,B 0,C 180,E1 -21313.603,E2 -21313.603} C_VEL
LIN {X 0,Y 197.847,Z 603.729,A -85,B 0,C 180,E1 -21317.689,E2 -21317.689} C_VEL
LIN {X 0,Y 197.282,Z 605.657,A -85,B 0,C 180,E1 -21321.803,E2 -21321.803} C_VEL
LIN {X 0,Y 197.239,Z 606.55,A -85,B 0,C 180,E1 -21326.092,E2 -21326.092} C_VEL
LIN {X 0,Y 197.377,Z 606.519,A -85,B 0,C 180,E1 -21329.995,E2 -21329.995} C_VEL
LIN {X 0,Y 197.244,Z 605.408,A -85,B 0,C 180,E1 -21334.081,E2 -21334.081} C_VEL
LIN {X 0,Y 197.285,Z 603.365,A -85,B 0,C 180,E1 -21338.187,E2 -21338.187} C_VEL
LIN {X 0,Y 197.822,Z 600.172,A -85,B 0,C 180,E1 -21342.302,E2 -21342.302} C_VEL
LIN {X 0,Y 199.11,Z 595.956,A -85,B 0,C 180,E1 -21346.396,E2 -21346.396} C_VEL
LIN {X 0,Y 201.017,Z 590.512,A -85,B 0,C 180,E1 -21350.458,E2 -21350.458} C_VEL
LIN {X 0,Y 203.762,Z 583.796,A -85,B 0,C 180,E1 -21354.443,E2 -21354.443} C_VEL
LIN {X 0,Y 207.301,Z 575.697,A -85,B 0,C 180,E1 -21358.329,E2 -21358.329} C_VEL
LIN {X 0,Y 211.724,Z 565.993,A -85,B 0,C 180,E1 -21362.073,E2 -21362.073} C_VEL
LIN {X 0,Y 216.283,Z 555.885,A -85,B 0,C 180,E1 -21365.217,E2 -21365.217} C_VEL
LIN {X 0,Y 221.426,Z 544.04,A -85,B 0,C 180,E1 -21368.23,E2 -21368.23} C_VEL
LIN {X 0,Y 226.722,Z 531.087,A -85,B 0,C 180,E1 -21370.9,E2 -21370.9} C_VEL
LIN {X 0,Y 231.302,Z 519.217,A -85,B 0,C 180,E1 -21372.9,E2 -21372.9} C_VEL
LIN {X 0,Y 236.301,Z 504.418,A -85,B 0,C 180,E1 -21374.932,E2 -21374.932} C_VEL
LIN {X 0,Y 240.299,Z 491.269,A -85,B 0,C 180,E1 -21376.366,E2 -21376.366} C_VEL
LIN {X 0,Y 244.389,Z 475.428,A -85,B 0,C 180,E1 -21377.766,E2 -21377.766} C_VEL
LIN {X 0,Y 247.848,Z 459.178,A -85,B 0,C 180,E1 -21378.86,E2 -21378.86} C_VEL
LIN {X 0,Y 250.615,Z 442.449,A -85,B 0,C 180,E1 -21379.677,E2 -21379.677} C_VEL
LIN {X 0,Y 252.36,Z 426.104,A -85,B 0,C 180,E1 -21380.228,E2 -21380.228} C_VEL
LIN {X 0,Y 259.664,Z 323.727,A -85,B 0,C 180,E1 -21382.912,E2 -21382.912} C_VEL
LIN {X 0,Y 253.011,Z 309.602,A -85,B 0,C 180,E1 -21385.214,E2 -21385.214} C_VEL
LIN {X 0,Y 246.057,Z 296.111,A -85,B 0,C 180,E1 -21387.783,E2 -21387.783} C_VEL
LIN {X 0,Y 239.026,Z 283.68,A -85,B 0,C 180,E1 -21390.602,E2 -21390.602} C_VEL
LIN {X 0,Y 231.523,Z 272.936,A -85,B 0,C 180,E1 -21393.836,E2 -21393.836} C_VEL
LIN {X 0,Y 224.949,Z 263.943,A -85,B 0,C 180,E1 -21397.029,E2 -21397.029} C_VEL
LIN {X 0,Y 221.545,Z 259.626,A -85,B 0,C 180,E1 -21398.826,E2 -21398.826} C_VEL
LIN {X 0,Y 218.609,Z 255.786,A -85,B 0,C 180,E1 -21400.517,E2 -21400.517} C_VEL
LIN {X 0,Y 217.531,Z 254.549,A -85,B 0,C 180,E1 -21401.152,E2 -21401.152} C_VEL
LIN {X 0,Y 214.767,Z 251.161,A -85,B 0,C 180,E1 -21402.873,E2 -21402.873} C_VEL
LIN {X 0,Y 213.786,Z 249.721,A -85,B 0,C 180,E1 -21403.53,E2 -21403.53} C_VEL
LIN {X 0,Y 211.071,Z 247.025,A -85,B 0,C 180,E1 -21405.355,E2 -21405.355} C_VEL
LIN {X 0,Y 209.73,Z 244.541,A -85,B 0,C 180,E1 -21406.435,E2 -21406.435} C_VEL
LIN {X 0,Y 207.005,Z 242.504,A -85,B 0,C 180,E1 -21408.496,E2 -21408.496} C_VEL
LIN {X 0,Y 205.38,Z 239.786,A -85,B 0,C 180,E1 -21409.963,E2 -21409.963} C_VEL
LIN {X 0,Y 205.042,Z 238.784,A -85,B 0,C 180,E1 -21410.33,E2 -21410.33} C_VEL
LIN {X 0,Y 201.975,Z 236.921,A -85,B 0,C 180,E1 -21413.131,E2 -21413.131} C_VEL
LIN {X 0,Y 200.461,Z 234.669,A -85,B 0,C 180,E1 -21414.91,E2 -21414.91} C_VEL
LIN {X 0,Y 199.996,Z 232.822,A -85,B 0,C 180,E1 -21415.719,E2 -21415.719} C_VEL
LIN {X 0,Y 200.453,Z 232.814,A -85,B 0,C 180,E1 -21420.001,E2 -21420.001} C_VEL
LIN {X 0,Y 199.998,Z 232.848,A -85,B 0,C 180,E1 -21424.031,E2 -21424.031} C_VEL
LIN {X 0,Y 200.064,Z 232.876,A -85,B 0,C 180,E1 -21428.079,E2 -21428.079} C_VEL
LIN {X 0,Y 199.847,Z 232.864,A -85,B 0,C 180,E1 -21432.182,E2 -21432.182} C_VEL
LIN {X 0,Y 199.78,Z 232.897,A -85,B 0,C 180,E1 -21436.347,E2 -21436.347} C_VEL
LIN {X 0,Y 199.681,Z 232.896,A -85,B 0,C 180,E1 -21440.608,E2 -21440.608} C_VEL
LIN {X 0,Y 199.653,Z 232.895,A -85,B 0,C 180,E1 -21444.988,E2 -21444.988} C_VEL
LIN {X 0,Y 199.652,Z 232.929,A -85,B 0,C 180,E1 -21449.527,E2 -21449.527} C_VEL
LIN {X 0,Y 199.659,Z 232.909,A -85,B 0,C 180,E1 -21451.575,E2 -21451.575} C_VEL
LIN {X 0,Y 200.269,Z 235.057,A -85,B 0,C 180,E1 -21452.514,E2 -21452.514} C_VEL
LIN {X 0,Y 201.934,Z 237.315,A -85,B 0,C 180,E1 -21454.385,E2 -21454.385} C_VEL
LIN {X 0,Y 204.813,Z 239.093,A -85,B 0,C 180,E1 -21457.061,E2 -21457.061} C_VEL
LIN {X 0,Y 206.267,Z 241.984,A -85,B 0,C 180,E1 -21458.471,E2 -21458.471} C_VEL
LIN {X 0,Y 208.678,Z 244.164,A -85,B 0,C 180,E1 -21460.356,E2 -21460.356} C_VEL
LIN {X 0,Y 209.635,Z 244.789,A -85,B 0,C 180,E1 -21461.052,E2 -21461.052} C_VEL
LIN {X 0,Y 211.385,Z 247.755,A -85,B 0,C 180,E1 -21462.427,E2 -21462.427} C_VEL
LIN {X 0,Y 214.145,Z 250.354,A -85,B 0,C 180,E1 -21464.25,E2 -21464.25} C_VEL
LIN {X 0,Y 216.547,Z 253.781,A -85,B 0,C 180,E1 -21465.813,E2 -21465.813} C_VEL
LIN {X 0,Y 218.44,Z 255.744,A -85,B 0,C 180,E1 -21466.93,E2 -21466.93} C_VEL
LIN {X 0,Y 221.292,Z 259.447,A -85,B 0,C 180,E1 -21468.57,E2 -21468.57} C_VEL
LIN {X 0,Y 222.821,Z 261.347,A -85,B 0,C 180,E1 -21469.394,E2 -21469.394} C_VEL
LIN {X 0,Y 226.801,Z 266.54,A -85,B 0,C 180,E1 -21471.443,E2 -21471.443} C_VEL
LIN {X 0,Y 229.995,Z 270.933,A -85,B 0,C 180,E1 -21472.985,E2 -21472.985} C_VEL
LIN {X 0,Y 235.389,Z 278.364,A -85,B 0,C 180,E1 -21475.4,E2 -21475.4} C_VEL
LIN {X 0,Y 243.16,Z 289.933,A -85,B 0,C 180,E1 -21478.557,E2 -21478.557} C_VEL
LIN {X 0,Y 252.474,Z 305.142,A -85,B 0,C 180,E1 -21481.953,E2 -21481.953} C_VEL
LIN {X 0,Y 259.769,Z 318.283,A -85,B 0,C 180,E1 -21484.395,E2 -21484.395} C_VEL
LIN {X 0,Y 252.243,Z 422.053,A -85,B 0,C 180,E1 -21487.136,E2 -21487.136} C_VEL
LIN {X 0,Y 250.086,Z 438.932,A -85,B 0,C 180,E1 -21487.834,E2 -21487.834} C_VEL
LIN {X 0,Y 247.292,Z 454.835,A -85,B 0,C 180,E1 -21488.76,E2 -21488.76} C_VEL
LIN {X 0,Y 243.836,Z 470.69,A -85,B 0,C 180,E1 -21489.99,E2 -21489.99} C_VEL
LIN {X 0,Y 240.015,Z 485.373,A -85,B 0,C 180,E1 -21491.437,E2 -21491.437} C_VEL
LIN {X 0,Y 235.624,Z 499.57,A -85,B 0,C 180,E1 -21493.166,E2 -21493.166} C_VEL
LIN {X 0,Y 230.818,Z 513.268,A -85,B 0,C 180,E1 -21495.231,E2 -21495.231} C_VEL
LIN {X 0,Y 226.178,Z 525.314,A -85,B 0,C 180,E1 -21497.442,E2 -21497.442} C_VEL
LIN {X 0,Y 221.139,Z 537.426,A -85,B 0,C 180,E1 -21500.139,E2 -21500.139} C_VEL
LIN {X 0,Y 216.505,Z 547.936,A -85,B 0,C 180,E1 -21503.013,E2 -21503.013} C_VEL
LIN {X 0,Y 212.043,Z 557.57,A -85,B 0,C 180,E1 -21506.204,E2 -21506.204} C_VEL
LIN {X 0,Y 207.713,Z 566.903,A -85,B 0,C 180,E1 -21510.005,E2 -21510.005} C_VEL
LIN {X 0,Y 204.18,Z 574.702,A -85,B 0,C 180,E1 -21513.952,E2 -21513.952} C_VEL
LIN {X 0,Y 201.389,Z 581.082,A -85,B 0,C 180,E1 -21518.029,E2 -21518.029} C_VEL
LIN {X 0,Y 199.415,Z 586.202,A -85,B 0,C 180,E1 -21522.212,E2 -21522.212} C_VEL
LIN {X 0,Y 197.969,Z 590.265,A -85,B 0,C 180,E1 -21526.557,E2 -21526.557} C_VEL
LIN {X 0,Y 197.096,Z 593.074,A -85,B 0,C 180,E1 -21530.895,E2 -21530.895} C_VEL
LIN {X 0,Y 196.741,Z 594.799,A -85,B 0,C 180,E1 -21535.387,E2 -21535.387} C_VEL
LIN {X 0,Y 196.755,Z 595.249,A -85,B 0,C 180,E1 -21537.673,E2 -21537.673} C_VEL
LIN {X 0,Y 196.964,Z 595.347,A -85,B 0,C 180,E1 -21541.088,E2 -21541.088} C_VEL
LIN {X 0,Y 197.523,Z 594.693,A -85,B 0,C 180,E1 -21545.077,E2 -21545.077} C_VEL
LIN {X 0,Y 198.76,Z 592.799,A -85,B 0,C 180,E1 -21549.533,E2 -21549.533} C_VEL
LIN {X 0,Y 200.98,Z 589.428,A -85,B 0,C 180,E1 -21554.381,E2 -21554.381} C_VEL
LIN {X 0,Y 203.303,Z 585.942,A -85,B 0,C 180,E1 -21557.988,E2 -21557.988} C_VEL
LIN {X 0,Y 207.079,Z 580.348,A -85,B 0,C 180,E1 -21562.344,E2 -21562.344} C_VEL
LIN {X 0,Y 211.47,Z 573.98,A -85,B 0,C 180,E1 -21566.191,E2 -21566.191} C_VEL
LIN {X 0,Y 216.958,Z 565.837,A -85,B 0,C 180,E1 -21570.062,E2 -21570.062} C_VEL
LIN {X 0,Y 222.521,Z 557.203,A -85,B 0,C 180,E1 -21573.307,E2 -21573.307} C_VEL
LIN {X 0,Y 228.956,Z 546.693,A -85,B 0,C 180,E1 -21576.48,E2 -21576.48} C_VEL
LIN {X 0,Y 235.739,Z 534.678,A -85,B 0,C 180,E1 -21579.39,E2 -21579.39} C_VEL
LIN {X 0,Y 241.74,Z 523.249,A -85,B 0,C 180,E1 -21581.605,E2 -21581.605} C_VEL
LIN {X 0,Y 247.647,Z 510.637,A -85,B 0,C 180,E1 -21583.618,E2 -21583.618} C_VEL
LIN {X 0,Y 253.331,Z 496.867,A -85,B 0,C 180,E1 -21585.397,E2 -21585.397} C_VEL
LIN {X 0,Y 258.474,Z 482.774,A -85,B 0,C 180,E1 -21586.851,E2 -21586.851} C_VEL
LIN {X 0,Y 263.096,Z 467.737,A -85,B 0,C 180,E1 -21588.105,E2 -21588.105} C_VEL
LIN {X 0,Y 267.177,Z 451.432,A -85,B 0,C 180,E1 -21589.15,E2 -21589.15} C_VEL
LIN {X 0,Y 270.333,Z 434.761,A -85,B 0,C 180,E1 -21589.933,E2 -21589.933} C_VEL
LIN {X 0,Y 272.546,Z 417.749,A -85,B 0,C 180,E1 -21590.48,E2 -21590.48} C_VEL
LIN {X 0,Y 280.458,Z 329.328,A -85,B 0,C 180,E1 -21592.688,E2 -21592.688} C_VEL
LIN {X 0,Y 276.191,Z 320.87,A -85,B 0,C 180,E1 -21595.155,E2 -21595.155} C_VEL
LIN {X 0,Y 271.688,Z 312.714,A -85,B 0,C 180,E1 -21598.222,E2 -21598.222} C_VEL
LIN {X 0,Y 268.663,Z 307.509,A -85,B 0,C 180,E1 -21600.722,E2 -21600.722} C_VEL
LIN {X 0,Y 266.055,Z 303.139,A -85,B 0,C 180,E1 -21603.429,E2 -21603.429} C_VEL
LIN {X 0,Y 263.859,Z 299.537,A -85,B 0,C 180,E1 -21606.528,E2 -21606.528} C_VEL
LIN {X 0,Y 261.936,Z 297.583,A -85,B 0,C 180,E1 -21611.57,E2 -21611.57} C_VEL
LIN {X 0,Y 261.844,Z 297.43,A -85,B 0,C 180,E1 -21614.268,E2 -21614.268} C_VEL
LIN {X 0,Y 261.926,Z 298.404,A -85,B 0,C 180,E1 -21615.541,E2 -21615.541} C_VEL
LIN {X 0,Y 262.105,Z 301.936,A -85,B 0,C 180,E1 -21617.563,E2 -21617.563} C_VEL
LIN {X 0,Y 262.761,Z 306.877,A -85,B 0,C 180,E1 -21619.956,E2 -21619.956} C_VEL
LIN {X 0,Y 263.192,Z 308.136,A -85,B 0,C 180,E1 -21620.779,E2 -21620.779} C_VEL
LIN {X 0,Y 265.182,Z 311.165,A -85,B 0,C 180,E1 -21623.424,E2 -21623.424} C_VEL
LIN {X 0,Y 267.557,Z 315.403,A -85,B 0,C 180,E1 -21625.911,E2 -21625.911} C_VEL
LIN {X 0,Y 269.567,Z 319.4,A -85,B 0,C 180,E1 -21627.672,E2 -21627.672} C_VEL
LIN {X 0,Y 272.327,Z 325.323,A -85,B 0,C 180,E1 -21629.811,E2 -21629.811} C_VEL
LIN {X 0,Y 275.515,Z 333.285,A -85,B 0,C 180,E1 -21632.025,E2 -21632.025} C_VEL
LIN {X 0,Y 276.833,Z 336.54,A -85,B 0,C 180,E1 -21632.841,E2 -21632.841} C_VEL
LIN {X 0,Y 267.988,Z 431.147,A -85,B 0,C 180,E1 -21635.227,E2 -21635.227} C_VEL
LIN {X 0,Y 265.078,Z 448.603,A -85,B 0,C 180,E1 -21635.837,E2 -21635.837} C_VEL
LIN {X 0,Y 261.505,Z 464.121,A -85,B 0,C 180,E1 -21636.589,E2 -21636.589} C_VEL
LIN {X 0,Y 257.133,Z 479.406,A -85,B 0,C 180,E1 -21637.565,E2 -21637.565} C_VEL
LIN {X 0,Y 252.295,Z 493.691,A -85,B 0,C 180,E1 -21638.738,E2 -21638.738} C_VEL
LIN {X 0,Y 245.886,Z 509.757,A -85,B 0,C 180,E1 -21640.444,E2 -21640.444} C_VEL
LIN {X 0,Y 239.18,Z 524.263,A -85,B 0,C 180,E1 -21642.413,E2 -21642.413} C_VEL
LIN {X 0,Y 232.329,Z 537.512,A -85,B 0,C 180,E1 -21644.69,E2 -21644.69} C_VEL
LIN {X 0,Y 225.38,Z 549.706,A -85,B 0,C 180,E1 -21647.291,E2 -21647.291} C_VEL
LIN {X 0,Y 218.268,Z 561.274,A -85,B 0,C 180,E1 -21650.401,E2 -21650.401} C_VEL
LIN {X 0,Y 211.654,Z 571.482,A -85,B 0,C 180,E1 -21653.882,E2 -21653.882} C_VEL
LIN {X 0,Y 206.61,Z 578.919,A -85,B 0,C 180,E1 -21657.022,E2 -21657.022} C_VEL
LIN {X 0,Y 201.697,Z 586.136,A -85,B 0,C 180,E1 -21660.798,E2 -21660.798} C_VEL
LIN {X 0,Y 197.673,Z 592.171,A -85,B 0,C 180,E1 -21664.741,E2 -21664.741} C_VEL
LIN {X 0,Y 193.94,Z 598.074,A -85,B 0,C 180,E1 -21669.859,E2 -21669.859} C_VEL
